C05494=1175.182,115.152,-52.912,-178.804,6.300,148.789
C05495=1175.178,115.401,-52.932,-178.801,6.302,148.788
C05496=1175.172,115.650,-52.951,-178.799,6.303,148.788
C05497=1175.168,115.900,-52.970,-178.796,6.304,148.787
C05498=1175.163,116.148,-52.989,-178.794,6.306,148.787
C05499=1175.158,116.398,-53.009,-178.790,6.307,148.786
C05500=1175.154,116.646,-53.028,-178.788,6.308,148.786
C05501=1175.149,116.897,-53.047,-178.786,6.310,148.785
C05502=1175.143,117.146,-53.066,-178.782,6.311,148.785
C05503=1175.139,117.395,-53.085,-178.780,6.312,148.784
C05504=1175.134,117.644,-53.105,-178.778,6.314,148.784
C05505=1175.129,117.893,-53.124,-178.775,6.316,148.784
C05506=1175.125,118.143,-53.143,-178.772,6.317,148.783
C05507=1175.120,118.391,-53.162,-178.770,6.318,148.783
C05508=1175.115,118.641,-53.182,-178.767,6.320,148.782
C05509=1175.110,118.890,-53.201,-178.764,6.322,148.782
C05510=1175.106,119.139,-53.220,-178.761,6.323,148.781
C05511=1175.101,119.389,-53.240,-178.759,6.324,148.781
C05512=1175.096,119.638,-53.259,-178.756,6.326,148.780
C05513=1175.091,119.887,-53.279,-178.753,6.327,148.780
C05514=1175.086,120.136,-53.298,-178.751,6.328,148.779
C05515=1175.082,120.385,-53.317,-178.748,6.330,148.779
C05516=1175.077,120.635,-53.337,-178.745,6.331,148.778
C05517=1175.071,120.884,-53.356,-178.743,6.333,148.778
C05518=1175.067,121.133,-53.376,-178.740,6.334,148.777
C05519=1175.062,121.382,-53.394,-178.737,6.335,148.777
C05520=1175.057,121.631,-53.414,-178.735,6.337,148.777
C05521=1175.053,121.880,-53.434,-178.732,6.339,148.776
C05522=1175.048,122.129,-53.454,-178.729,6.339,148.776
C05523=1175.043,122.379,-53.473,-178.727,6.341,148.775
C05524=1175.039,122.628,-53.492,-178.724,6.343,148.775
C05525=1175.033,122.877,-53.512,-178.721,6.345,148.774
C05526=1175.029,123.126,-53.531,-178.719,6.345,148.774
C05527=1175.024,123.376,-53.551,-178.716,6.347,148.773
C05528=1175.019,123.624,-53.571,-178.713,6.349,148.773
C05529=1175.014,123.874,-53.591,-178.711,6.350,148.773
C05530=1175.009,124.123,-53.610,-178.708,6.352,148.772
C05531=1175.004,124.372,-53.630,-178.705,6.353,148.772
C05532=1175.000,124.621,-53.649,-178.703,6.354,148.771
C05533=1174.996,124.870,-53.669,-178.700,6.356,148.771
C05534=1174.990,125.119,-53.688,-178.697,6.358,148.770
C05535=1174.986,125.369,-53.708,-178.694,6.358,148.770
C05536=1174.981,125.618,-53.728,-178.692,6.360,148.769
C05537=1174.976,125.867,-53.748,-178.689,6.362,148.769
C05538=1174.971,126.116,-53.767,-178.686,6.364,148.769
C05539=1174.966,126.366,-53.787,-178.684,6.365,148.768
C05540=1174.962,126.615,-53.807,-178.681,6.366,148.768
C05541=1174.957,126.864,-53.827,-178.678,6.368,148.767
C05542=1174.952,127.113,-53.846,-178.676,6.369,148.767
C05543=1174.947,127.363,-53.866,-178.673,6.371,148.766
C05544=1174.943,127.612,-53.886,-178.670,6.372,148.766
C05545=1174.937,127.861,-53.906,-178.668,6.374,148.765
C05546=1174.933,128.110,-53.926,-178.665,6.375,148.765
C05547=1174.928,128.359,-53.946,-178.662,6.377,148.765
C05548=1174.923,128.609,-53.965,-178.660,6.379,148.764
C05549=1174.918,128.857,-53.985,-178.657,6.379,148.763
C05550=1174.914,129.106,-54.005,-178.654,6.381,148.763
C05551=1174.909,129.356,-54.025,-178.652,6.383,148.763
C05552=1174.904,129.605,-54.045,-178.649,6.385,148.762
C05553=1174.900,129.855,-54.065,-178.646,6.386,148.762
C05554=1174.895,130.103,-54.085,-178.644,6.387,148.761
C05555=1174.890,130.352,-54.104,-178.641,6.389,148.761
C05556=1174.885,130.601,-54.125,-178.638,6.390,148.760
C05557=1174.881,130.851,-54.144,-178.635,6.392,148.760
C05558=1174.876,131.099,-54.164,-178.633,6.394,148.760
C05559=1174.871,131.349,-54.184,-178.631,6.395,148.759
C05560=1174.866,131.598,-54.204,-178.627,6.396,148.759
C05561=1174.861,131.848,-54.225,-178.625,6.398,148.758
C05562=1174.856,132.116,-54.247,-178.622,6.400,148.758
C05563=1174.851,132.385,-54.268,-178.619,6.401,148.757
C05564=1174.846,132.653,-54.289,-178.616,6.403,148.757
C05565=1174.841,132.921,-54.311,-178.613,6.404,148.757
C05566=1174.836,133.171,-54.331,-178.611,6.406,148.756
C05567=1174.831,133.420,-54.352,-178.608,6.408,148.756
C05568=1174.826,133.669,-54.371,-178.605,6.409,148.755
C05569=1174.821,133.918,-54.391,-178.603,6.410,148.755
C05570=1174.817,134.167,-54.412,-178.600,6.412,148.754
C05571=1174.812,134.416,-54.431,-178.597,6.414,148.754
C05572=1174.807,134.666,-54.452,-178.595,6.415,148.754
C05573=1174.803,134.915,-54.473,-178.591,6.417,148.753
C05574=1174.798,135.164,-54.492,-178.589,6.419,148.753
C05575=1174.794,135.413,-54.513,-178.586,6.420,148.752
C05576=1174.788,135.661,-54.533,-178.584,6.421,148.752
C05577=1174.783,135.911,-54.553,-178.581,6.423,148.751
C05578=1174.779,136.160,-54.573,-178.579,6.425,148.751
C05579=1174.774,136.409,-54.594,-178.575,6.426,148.750
C05580=1174.769,136.659,-54.613,-178.573,6.428,148.750
C05581=1174.764,136.908,-54.634,-178.570,6.430,148.750
C05582=1174.760,137.157,-54.655,-178.568,6.431,148.749
C05583=1174.755,137.406,-54.675,-178.565,6.432,148.749
C05584=1174.751,137.655,-54.695,-178.562,6.434,148.748
C05585=1174.745,137.905,-54.716,-178.560,6.436,148.748
C05586=1174.741,138.154,-54.736,-178.557,6.437,148.747
C05587=1174.737,138.403,-54.756,-178.554,6.439,148.747
C05588=1174.731,138.652,-54.777,-178.551,6.441,148.747
C05589=1174.726,138.901,-54.797,-178.549,6.442,148.746
C05590=1174.722,139.150,-54.817,-178.546,6.443,148.746
C05591=1174.716,139.399,-54.838,-178.544,6.445,148.745
C05592=1174.712,139.648,-54.858,-178.541,6.447,148.745
C05593=1174.708,139.897,-54.879,-178.538,6.448,148.744
C05594=1174.702,140.146,-54.900,-178.535,6.450,148.744
C05595=1174.698,140.395,-54.920,-178.532,6.452,148.744
C05596=1174.693,140.645,-54.940,-178.530,6.453,148.743
C05597=1174.688,140.894,-54.961,-178.528,6.454,148.743
C05598=1174.684,141.143,-54.981,-178.525,6.456,148.743
C05599=1174.679,141.392,-55.002,-178.522,6.458,148.742
C05600=1174.674,141.641,-55.023,-178.519,6.460,148.742
C05601=1174.670,141.890,-55.043,-178.517,6.461,148.741
C05602=1174.664,142.139,-55.064,-178.514,6.463,148.741
C05603=1174.660,142.388,-55.084,-178.511,6.465,148.740
C05604=1174.655,142.637,-55.105,-178.508,6.466,148.740
C05605=1174.650,142.886,-55.126,-178.505,6.468,148.740
C05606=1174.646,143.135,-55.146,-178.503,6.469,148.739
C05607=1174.641,143.385,-55.167,-178.501,6.471,148.739
C05608=1174.636,143.634,-55.187,-178.498,6.472,148.738
C05609=1174.631,143.883,-55.208,-178.495,6.474,148.738
C05610=1174.627,144.132,-55.229,-178.493,6.476,148.738
C05611=1174.622,144.382,-55.250,-178.489,6.477,148.737
C05612=1174.618,144.631,-55.270,-178.487,6.479,148.737
C05613=1174.612,144.880,-55.291,-178.484,6.481,148.736
C05614=1174.608,145.128,-55.312,-178.481,6.483,148.736
C05615=1174.603,145.378,-55.333,-178.479,6.484,148.736
C05616=1174.599,145.626,-55.354,-178.477,6.485,148.735
C05617=1174.594,145.876,-55.375,-178.474,6.487,148.735
C05618=1174.589,146.125,-55.395,-178.471,6.489,148.734
C05619=1174.584,146.374,-55.416,-178.468,6.491,148.734
C05620=1174.579,146.623,-55.436,-178.466,6.492,148.734
C05621=1174.574,146.872,-55.457,-178.463,6.494,148.733
C05622=1174.571,147.121,-55.479,-178.460,6.495,148.733
C05623=1174.566,147.370,-55.500,-178.457,6.497,148.732
C05624=1174.561,147.619,-55.520,-178.454,6.499,148.732
C05625=1174.556,147.869,-55.541,-178.452,6.501,148.731
C05626=1174.551,148.118,-55.562,-178.449,6.502,148.731
C05627=1174.547,148.366,-55.583,-178.446,6.504,148.731
C05628=1174.542,148.615,-55.604,-178.444,6.506,148.730
C05629=1174.537,148.864,-55.624,-178.442,6.507,148.730
C05630=1174.532,149.114,-55.645,-178.439,6.509,148.730
C05631=1174.528,149.363,-55.668,-178.436,6.510,148.729
C05632=1174.523,149.612,-55.688,-178.433,6.512,148.729
C05633=1174.518,149.861,-55.709,-178.431,6.514,148.728
C05634=1174.514,150.110,-55.730,-178.428,6.516,148.728
C05635=1174.509,150.359,-55.751,-178.425,6.517,148.727
C05636=1174.504,150.608,-55.772,-178.422,6.519,148.727
C05637=1174.500,150.857,-55.793,-178.420,6.521,148.727
C05638=1174.495,151.106,-55.814,-178.417,6.522,148.726
C05639=1174.490,151.356,-55.835,-178.414,6.524,148.726
C05640=1174.485,151.604,-55.857,-178.411,6.526,148.726
C05641=1174.480,151.853,-55.877,-178.409,6.528,148.725
C05642=1174.476,152.103,-55.899,-178.406,6.529,148.725
C05643=1174.471,152.352,-55.920,-178.403,6.531,148.724
C05644=1174.466,152.601,-55.941,-178.401,6.533,148.724
C05645=1174.462,152.849,-55.962,-178.398,6.535,148.724
C05646=1174.456,153.099,-55.983,-178.395,6.536,148.723
C05647=1174.452,153.348,-56.005,-178.393,6.538,148.723
C05648=1174.448,153.597,-56.026,-178.390,6.540,148.722
C05649=1174.443,153.846,-56.047,-178.387,6.542,148.722
C05650=1174.438,154.095,-56.068,-178.385,6.543,148.722
C05651=1174.433,154.343,-56.090,-178.382,6.544,148.721
C05652=1174.429,154.593,-56.111,-178.380,6.546,148.721
C05653=1174.424,154.842,-56.133,-178.377,6.548,148.721
C05654=1174.419,155.091,-56.153,-178.374,6.550,148.720
C05655=1174.414,155.340,-56.175,-178.372,6.551,148.720
C05656=1174.409,155.590,-56.197,-178.369,6.553,148.719
C05657=1174.405,155.838,-56.218,-178.366,6.555,148.719
C05658=1174.400,156.087,-56.239,-178.363,6.556,148.718
C05659=1174.396,156.337,-56.261,-178.360,6.558,148.718
C05660=1174.391,156.586,-56.282,-178.358,6.560,148.718
C05661=1174.386,156.834,-56.303,-178.355,6.562,148.717
C05662=1174.381,157.083,-56.325,-178.352,6.563,148.717
C05663=1174.377,157.333,-56.346,-178.350,6.565,148.717
C05664=1174.372,157.581,-56.367,-178.347,6.567,148.716
C05665=1174.367,157.830,-56.389,-178.344,6.569,148.716
C05666=1174.362,158.099,-56.412,-178.341,6.571,148.716
C05667=1174.357,158.368,-56.435,-178.338,6.573,148.715
C05668=1174.352,158.638,-56.459,-178.336,6.575,148.715
C05669=1174.347,158.906,-56.482,-178.333,6.576,148.714
C05670=1174.342,159.156,-56.503,-178.330,6.578,148.714
C05671=1174.338,159.405,-56.525,-178.328,6.580,148.714
C05672=1174.333,159.653,-56.547,-178.325,6.582,148.713
C05673=1174.328,159.902,-56.568,-178.322,6.583,148.713
C05674=1174.324,160.152,-56.590,-178.320,6.585,148.713
C05675=1174.319,160.401,-56.611,-178.317,6.587,148.712
C05676=1174.314,160.649,-56.633,-178.314,6.589,148.712
C05677=1174.310,160.899,-56.655,-178.311,6.590,148.711
C05678=1174.305,161.147,-56.677,-178.309,6.592,148.711
C05679=1174.300,161.397,-56.698,-178.306,6.594,148.711
C05680=1174.295,161.646,-56.720,-178.303,6.596,148.710
C05681=1174.290,161.895,-56.742,-178.301,6.598,148.710
C05682=1174.286,162.144,-56.764,-178.298,6.599,148.710
C05683=1174.281,162.393,-56.785,-178.295,6.602,148.709
C05684=1174.277,162.642,-56.807,-178.292,6.604,148.709
C05685=1174.272,162.891,-56.828,-178.289,6.605,148.708
C05686=1174.267,163.140,-56.850,-178.287,6.607,148.708
C05687=1174.263,163.389,-56.872,-178.284,6.609,148.708
C05688=1174.258,163.638,-56.894,-178.281,6.611,148.707
C05689=1174.253,163.887,-56.916,-178.279,6.612,148.707
C05690=1174.249,164.136,-56.937,-178.276,6.614,148.707
C05691=1174.244,164.384,-56.959,-178.273,6.616,148.706
C05692=1174.239,164.634,-56.981,-178.271,6.618,148.706
C05693=1174.235,164.882,-57.003,-178.268,6.619,148.705
C05694=1174.230,165.132,-57.025,-178.265,6.621,148.705
C05695=1174.225,165.380,-57.047,-178.263,6.623,148.705
C05696=1174.221,165.630,-57.069,-178.260,6.625,148.704
C05697=1174.216,165.878,-57.090,-178.257,6.627,148.704
C05698=1174.211,166.128,-57.113,-178.254,6.628,148.704
C05699=1174.206,166.377,-57.135,-178.252,6.630,148.703
C05700=1174.202,166.626,-57.157,-178.249,6.632,148.703
C05701=1174.197,166.875,-57.178,-178.247,6.634,148.703
C05702=1174.193,167.124,-57.200,-178.244,6.636,148.702
C05703=1174.188,167.373,-57.222,-178.242,6.637,148.702
C05704=1174.184,167.622,-57.244,-178.238,6.640,148.702
C05705=1174.178,167.871,-57.266,-178.236,6.642,148.701
C05706=1174.174,168.120,-57.288,-178.233,6.644,148.701
C05707=1174.169,168.369,-57.310,-178.230,6.645,148.701
C05708=1174.165,168.618,-57.333,-178.228,6.647,148.700
C05709=1174.160,168.866,-57.355,-178.225,6.649,148.700
C05710=1174.155,169.116,-57.377,-178.222,6.651,148.699
C05711=1174.150,169.365,-57.399,-178.219,6.652,148.699
C05712=1174.146,169.614,-57.421,-178.217,6.654,148.699
C05713=1174.141,169.863,-57.443,-178.214,6.656,148.698
C05714=1174.137,170.112,-57.466,-178.211,6.658,148.698
C05715=1174.132,170.360,-57.488,-178.209,6.659,148.698
C05716=1174.127,170.610,-57.510,-178.207,6.662,148.697
C05717=1174.123,170.858,-57.531,-178.203,6.664,148.697
C05718=1174.118,171.107,-57.555,-178.201,6.666,148.697
C05719=1174.113,171.356,-57.576,-178.198,6.668,148.696
C05720=1174.109,171.605,-57.598,-178.195,6.669,148.696
C05721=1174.104,171.855,-57.621,-178.193,6.671,148.696
C05722=1174.099,172.103,-57.644,-178.190,6.673,148.695
C05723=1174.095,172.352,-57.666,-178.187,6.675,148.695
C05724=1174.089,172.601,-57.688,-178.185,6.676,148.695
C05725=1174.085,172.850,-57.711,-178.182,6.678,148.694
C05726=1174.081,173.099,-57.733,-178.179,6.680,148.694
C05727=1174.075,173.348,-57.755,-178.176,6.683,148.694
C05728=1174.072,173.597,-57.778,-178.174,6.685,148.693
C05729=1174.067,173.846,-57.799,-178.171,6.686,148.693
C05730=1174.062,174.095,-57.822,-178.168,6.688,148.693
C05731=1174.058,174.344,-57.845,-178.166,6.690,148.692
C05732=1174.053,174.593,-57.866,-178.163,6.692,148.692
C05733=1174.048,174.842,-57.890,-178.160,6.694,148.692
C05734=1174.044,175.091,-57.912,-178.158,6.695,148.691
C05735=1174.038,175.340,-57.934,-178.155,6.697,148.691
C05736=1174.034,175.589,-57.957,-178.152,6.700,148.691
C05737=1174.029,175.837,-57.979,-178.149,6.702,148.690
C05738=1174.025,176.086,-58.002,-178.147,6.704,148.690
C05739=1174.020,176.336,-58.024,-178.144,6.705,148.690
C05740=1174.015,176.584,-58.047,-178.141,6.707,148.689
C05741=1174.011,176.833,-58.069,-178.139,6.709,148.689
C05742=1174.006,177.082,-58.092,-178.136,6.711,148.688
C05743=1174.002,177.332,-58.114,-178.133,6.713,148.688
C05744=1173.997,177.580,-58.137,-178.131,6.715,148.688
C05745=1173.992,177.829,-58.159,-178.128,6.717,148.688
C05746=1173.988,178.078,-58.182,-178.125,6.719,148.687
C05747=1173.983,178.326,-58.205,-178.123,6.721,148.687
C05748=1173.979,178.576,-58.227,-178.120,6.722,148.687
C05749=1173.974,178.825,-58.251,-178.117,6.724,148.686
C05750=1173.969,179.074,-58.273,-178.114,6.727,148.686
C05751=1173.965,179.322,-58.296,-178.111,6.729,148.685
C05752=1173.960,179.571,-58.319,-178.109,6.731,148.685
C05753=1173.956,179.821,-58.341,-178.106,6.732,148.685
C05754=1173.950,180.069,-58.364,-178.104,6.734,148.685
C05755=1173.946,180.318,-58.387,-178.101,6.736,148.684
C05756=1173.941,180.568,-58.410,-178.098,6.738,148.684
C05757=1173.937,180.816,-58.432,-178.095,6.740,148.684
C05758=1173.932,181.065,-58.455,-178.093,6.742,148.683
C05759=1173.928,181.314,-58.477,-178.090,6.744,148.683
C05760=1173.923,181.563,-58.501,-178.088,6.746,148.683
C05761=1173.918,181.812,-58.524,-178.085,6.748,148.682
C05762=1173.914,182.060,-58.546,-178.082,6.750,148.682
C05763=1173.909,182.310,-58.569,-178.079,6.752,148.682
C05764=1173.905,182.558,-58.592,-178.077,6.754,148.682
C05765=1173.900,182.807,-58.615,-178.074,6.756,148.681
C05766=1173.895,183.056,-58.639,-178.071,6.758,148.681
C05767=1173.891,183.304,-58.661,-178.069,6.760,148.680
C05768=1173.886,183.554,-58.684,-178.066,6.761,148.680
C05769=1173.881,183.803,-58.707,-178.063,6.764,148.680
C05770=1173.877,184.073,-58.731,-178.060,6.766,148.679
C05771=1173.871,184.342,-58.756,-178.057,6.768,148.679
C05772=1173.866,184.612,-58.781,-178.054,6.770,148.679
C05773=1173.862,184.881,-58.807,-178.052,6.772,148.679
C05774=1173.857,185.130,-58.830,-178.049,6.775,148.678
C05775=1173.852,185.380,-58.853,-178.046,6.777,148.678
C05776=1173.848,185.628,-58.875,-178.043,6.778,148.678
C05777=1173.843,185.877,-58.898,-178.041,6.780,148.677
C05778=1173.838,186.126,-58.922,-178.038,6.782,148.677
C05779=1173.833,186.375,-58.945,-178.035,6.785,148.677
C05780=1173.829,186.623,-58.968,-178.033,6.787,148.676
C05781=1173.825,186.872,-58.991,-178.030,6.788,148.676
C05782=1173.820,187.122,-59.015,-178.027,6.790,148.676
C05783=1173.815,187.371,-59.038,-178.025,6.792,148.676
C05784=1173.811,187.619,-59.061,-178.022,6.795,148.675
C05785=1173.806,187.868,-59.084,-178.019,6.797,148.675
C05786=1173.801,188.117,-59.107,-178.016,6.798,148.674
C05787=1173.797,188.366,-59.130,-178.014,6.800,148.674
C05788=1173.792,188.615,-59.154,-178.011,6.803,148.674
C05789=1173.787,188.864,-59.177,-178.008,6.805,148.674
C05790=1173.783,189.112,-59.200,-178.006,6.807,148.673
C05791=1173.779,189.361,-59.223,-178.003,6.808,148.673
C05792=1173.774,189.611,-59.247,-178.000,6.810,148.673
C05793=1173.769,189.859,-59.271,-177.997,6.813,148.672
C05794=1173.765,190.108,-59.294,-177.995,6.815,148.672
C05795=1173.760,190.357,-59.317,-177.992,6.817,148.672
C05796=1173.755,190.605,-59.340,-177.989,6.819,148.671
C05797=1173.751,190.854,-59.363,-177.987,6.821,148.671
C05798=1173.746,191.103,-59.387,-177.984,6.823,148.671
C05799=1173.741,191.352,-59.410,-177.981,6.825,148.671
C05800=1173.737,191.601,-59.434,-177.979,6.827,148.670
C05801=1173.732,191.850,-59.457,-177.976,6.829,148.670
C05802=1173.728,192.099,-59.481,-177.973,6.832,148.670
C05803=1173.723,192.348,-59.504,-177.971,6.833,148.669
C05804=1173.718,192.596,-59.528,-177.968,6.835,148.669
C05805=1173.714,192.845,-59.551,-177.966,6.837,148.669
C05806=1173.709,193.094,-59.575,-177.962,6.840,148.669
C05807=1173.704,193.343,-59.598,-177.960,6.842,148.668
C05808=1173.700,193.592,-59.622,-177.957,6.843,148.668
C05809=1173.695,193.841,-59.646,-177.955,6.845,148.668
C05810=1173.691,194.090,-59.669,-177.952,6.848,148.667
C05811=1173.686,194.339,-59.692,-177.949,6.850,148.667
C05812=1173.682,194.587,-59.716,-177.946,6.852,148.667
C05813=1173.677,194.836,-59.740,-177.944,6.854,148.667
C05814=1173.672,195.084,-59.764,-177.941,6.856,148.666
C05815=1173.668,195.334,-59.787,-177.938,6.858,148.666
C05816=1173.663,195.583,-59.811,-177.936,6.860,148.666
C05817=1173.659,195.831,-59.835,-177.933,6.863,148.665
C05818=1173.654,196.080,-59.858,-177.930,6.865,148.665
C05819=1173.649,196.329,-59.881,-177.927,6.866,148.665
C05820=1173.645,196.577,-59.905,-177.925,6.868,148.664
C05821=1173.641,196.827,-59.929,-177.922,6.871,148.664
C05822=1173.636,197.076,-59.953,-177.919,6.873,148.664
C05823=1173.632,197.325,-59.977,-177.917,6.875,148.664
C05824=1173.627,197.573,-60.001,-177.914,6.877,148.664
C05825=1173.623,197.822,-60.024,-177.911,6.879,148.663
C05826=1173.617,198.071,-60.049,-177.909,6.881,148.663
C05827=1173.613,198.320,-60.072,-177.906,6.883,148.662
C05828=1173.608,198.568,-60.096,-177.903,6.886,148.662
C05829=1173.604,198.817,-60.119,-177.900,6.888,148.662
C05830=1173.599,199.066,-60.144,-177.898,6.889,148.662
C05831=1173.595,199.315,-60.167,-177.896,6.892,148.662
C05832=1173.591,199.564,-60.191,-177.892,6.894,148.661
C05833=1173.585,199.813,-60.215,-177.890,6.896,148.661
C05834=1173.581,200.062,-60.239,-177.887,6.898,148.661
C05835=1173.576,200.310,-60.263,-177.884,6.901,148.660
C05836=1173.572,200.559,-60.287,-177.882,6.903,148.660
C05837=1173.567,200.807,-60.311,-177.879,6.904,148.660
C05838=1173.563,201.056,-60.335,-177.876,6.907,148.660
C05839=1173.558,201.306,-60.359,-177.873,6.909,148.659
C05840=1173.554,201.554,-60.383,-177.871,6.911,148.659
C05841=1173.549,201.803,-60.407,-177.869,6.913,148.659
C05842=1173.545,202.052,-60.431,-177.865,6.916,148.659
C05843=1173.540,202.300,-60.455,-177.863,6.917,148.658
C05844=1173.535,202.549,-60.480,-177.860,6.919,148.658
C05845=1173.531,202.799,-60.503,-177.857,6.922,148.658
C05846=1173.527,203.047,-60.527,-177.855,6.924,148.657
C05847=1173.522,203.296,-60.552,-177.852,6.926,148.657
C05848=1173.517,203.544,-60.576,-177.849,6.929,148.657
C05849=1173.512,203.793,-60.599,-177.846,6.930,148.657
C05850=1173.509,204.042,-60.624,-177.844,6.932,148.656
C05851=1173.504,204.291,-60.649,-177.841,6.935,148.656
C05852=1173.499,204.539,-60.673,-177.838,6.937,148.656
C05853=1173.495,204.788,-60.697,-177.836,6.939,148.656
C05854=1173.489,205.037,-60.721,-177.833,6.942,148.655
C05855=1173.485,205.286,-60.745,-177.830,6.943,148.655
C05856=1173.481,205.535,-60.769,-177.828,6.946,148.655
C05857=1173.476,205.783,-60.794,-177.825,6.948,148.655
C05858=1173.472,206.032,-60.818,-177.822,6.950,148.654
C05859=1173.467,206.281,-60.843,-177.820,6.952,148.654
C05860=1173.463,206.530,-60.867,-177.817,6.955,148.654
C05861=1173.458,206.779,-60.890,-177.814,6.957,148.654
C05862=1173.453,207.027,-60.915,-177.812,6.959,148.653
C05863=1173.449,207.277,-60.939,-177.809,6.961,148.653
C05864=1173.444,207.525,-60.964,-177.806,6.963,148.653
C05865=1173.439,207.774,-60.988,-177.804,6.965,148.653
C05866=1173.436,208.023,-61.013,-177.800,6.968,148.652
C05867=1173.431,208.272,-61.037,-177.798,6.970,148.652
C05868=1173.426,208.520,-61.061,-177.796,6.972,148.652
C05869=1173.421,208.769,-61.086,-177.792,6.974,148.651
C05870=1173.417,209.018,-61.111,-177.790,6.976,148.651
C05871=1173.412,209.267,-61.135,-177.787,6.979,148.651
C05872=1173.408,209.515,-61.159,-177.785,6.981,148.651
C05873=1173.403,209.764,-61.184,-177.782,6.983,148.651
C05874=1173.398,210.035,-61.211,-177.779,6.985,148.650
C05875=1173.393,210.305,-61.238,-177.776,6.988,148.650
C05876=1173.389,210.575,-61.264,-177.773,6.990,148.650
C05877=1173.384,210.845,-61.291,-177.770,6.993,148.649
C05878=1173.379,211.094,-61.316,-177.768,6.995,148.649
C05879=1173.375,211.343,-61.340,-177.765,6.998,148.649
C05880=1173.370,211.592,-61.365,-177.762,6.999,148.649
C05881=1173.365,211.841,-61.389,-177.760,7.001,148.649
C05882=1173.361,212.090,-61.414,-177.757,7.004,148.648
C05883=1173.356,212.338,-61.439,-177.754,7.006,148.648
C05884=1173.352,212.587,-61.464,-177.751,7.009,148.648
C05885=1173.347,212.836,-61.488,-177.749,7.011,148.648
C05886=1173.343,213.084,-61.512,-177.746,7.013,148.647
C05887=1173.338,213.334,-61.537,-177.743,7.015,148.647
C05888=1173.333,213.582,-61.563,-177.741,7.017,148.647
C05889=1173.329,213.830,-61.587,-177.738,7.020,148.647
C05890=1173.325,214.080,-61.612,-177.735,7.022,148.646
C05891=1173.319,214.328,-61.637,-177.733,7.024,148.646
C05892=1173.316,214.577,-61.662,-177.730,7.027,148.646
C05893=1173.311,214.826,-61.686,-177.727,7.029,148.646
C05894=1173.307,215.075,-61.711,-177.724,7.031,148.645
C05895=1173.302,215.323,-61.736,-177.722,7.033,148.645
C05896=1173.297,215.571,-61.761,-177.719,7.035,148.645
C05897=1173.293,215.821,-61.785,-177.716,7.038,148.645
C05898=1173.288,216.069,-61.811,-177.714,7.040,148.645
C05899=1173.284,216.318,-61.836,-177.711,7.043,148.644
C05900=1173.279,216.567,-61.860,-177.709,7.045,148.644
C05901=1173.275,216.815,-61.886,-177.706,7.047,148.644
C05902=1173.270,217.064,-61.910,-177.703,7.049,148.644
C05903=1173.266,217.313,-61.936,-177.700,7.051,148.643
C05904=1173.262,217.561,-61.960,-177.697,7.054,148.643
C05905=1173.257,217.810,-61.986,-177.695,7.056,148.643
C05906=1173.252,218.059,-62.010,-177.692,7.059,148.643
C05907=1173.248,218.308,-62.036,-177.690,7.061,148.643
C05908=1173.244,218.556,-62.060,-177.687,7.063,148.642
C05909=1173.239,218.805,-62.085,-177.684,7.066,148.642
C05910=1173.234,219.054,-62.111,-177.682,7.067,148.642
C05911=1173.230,219.303,-62.136,-177.678,7.070,148.641
C05912=1173.226,219.551,-62.161,-177.676,7.072,148.641
C05913=1173.221,219.800,-62.186,-177.673,7.075,148.641
C05914=1173.216,220.048,-62.211,-177.671,7.077,148.641
C05915=1173.212,220.297,-62.237,-177.668,7.079,148.641
C05916=1173.207,220.546,-62.261,-177.665,7.082,148.641
C05917=1173.203,220.795,-62.287,-177.663,7.083,148.640
C05918=1173.198,221.043,-62.311,-177.660,7.086,148.640
C05919=1173.194,221.292,-62.337,-177.657,7.088,148.640
C05920=1173.189,221.540,-62.362,-177.654,7.091,148.640
C05921=1173.185,221.789,-62.387,-177.652,7.093,148.639
C05922=1173.180,222.038,-62.413,-177.649,7.096,148.639
C05923=1173.176,222.286,-62.439,-177.646,7.098,148.639
C05924=1173.171,222.536,-62.464,-177.644,7.101,148.639
C05925=1173.166,222.784,-62.489,-177.641,7.102,148.639
C05926=1173.163,223.032,-62.514,-177.639,7.104,148.638
C05927=1173.158,223.281,-62.539,-177.635,7.107,148.638
C05928=1173.153,223.530,-62.565,-177.633,7.109,148.638
C05929=1173.149,223.779,-62.590,-177.630,7.112,148.638
C05930=1173.144,224.027,-62.616,-177.628,7.114,148.638
C05931=1173.140,224.276,-62.641,-177.625,7.117,148.637
C05932=1173.136,224.525,-62.666,-177.622,7.119,148.637
C05933=1173.131,224.773,-62.692,-177.619,7.121,148.637
C05934=1173.127,225.022,-62.718,-177.617,7.123,148.637
C05935=1173.122,225.270,-62.743,-177.614,7.126,148.636
C05936=1173.117,225.519,-62.768,-177.612,7.128,148.636
C05937=1173.113,225.768,-62.794,-177.608,7.131,148.636
C05938=1173.108,226.016,-62.819,-177.606,7.133,148.636
C05939=1173.104,226.265,-62.845,-177.603,7.136,148.636
C05940=1173.100,226.514,-62.871,-177.601,7.138,148.636
C05941=1173.095,226.762,-62.896,-177.598,7.140,148.635
C05942=1173.091,227.011,-62.922,-177.595,7.142,148.635
C05943=1173.086,227.260,-62.947,-177.592,7.145,148.635
C05944=1173.081,227.508,-62.972,-177.590,7.147,148.635
C05945=1173.077,227.757,-62.998,-177.587,7.150,148.635
C05946=1173.073,228.006,-63.024,-177.585,7.152,148.634
C05947=1173.068,228.254,-63.049,-177.582,7.155,148.634
C05948=1173.063,228.503,-63.075,-177.579,7.157,148.634
C05949=1173.059,228.752,-63.101,-177.576,7.160,148.634
C05950=1173.054,229.000,-63.127,-177.574,7.162,148.633
C05951=1173.050,229.249,-63.152,-177.571,7.164,148.633
C05952=1173.046,229.498,-63.178,-177.568,7.166,148.633
C05953=1173.041,229.746,-63.204,-177.566,7.169,148.633
C05954=1173.036,229.995,-63.229,-177.563,7.171,148.633
C05955=1173.032,230.243,-63.255,-177.560,7.174,148.633
C05956=1173.027,230.493,-63.281,-177.558,7.176,148.632
C05957=1173.023,230.741,-63.307,-177.555,7.179,148.632
C05958=1173.018,230.989,-63.332,-177.553,7.181,148.632
C05959=1173.014,231.238,-63.359,-177.549,7.183,148.632
C05960=1173.010,231.486,-63.385,-177.547,7.186,148.632
C05961=1173.006,231.735,-63.410,-177.544,7.189,148.632
C05962=1173.000,231.984,-63.436,-177.542,7.190,148.631
C05963=1172.996,232.232,-63.462,-177.539,7.193,148.631
C05964=1172.992,232.481,-63.488,-177.536,7.195,148.631
C05965=1172.988,232.730,-63.514,-177.534,7.198,148.631
C05966=1172.982,232.978,-63.540,-177.531,7.200,148.631
C05967=1172.978,233.227,-63.566,-177.528,7.203,148.630
C05968=1172.974,233.475,-63.592,-177.526,7.205,148.630
C05969=1172.970,233.724,-63.618,-177.523,7.208,148.630
C05970=1172.965,233.973,-63.645,-177.520,7.211,148.630
C05971=1172.960,234.221,-63.670,-177.518,7.213,148.630
C05972=1172.956,234.470,-63.696,-177.515,7.215,148.630
C05973=1172.952,234.718,-63.722,-177.512,7.217,148.629
C05974=1172.947,234.967,-63.749,-177.509,7.220,148.629
C05975=1172.943,235.216,-63.774,-177.507,7.222,148.629
C05976=1172.939,235.465,-63.800,-177.504,7.225,148.629
C05977=1172.933,235.712,-63.827,-177.502,7.227,148.629
C05978=1172.929,235.984,-63.855,-177.499,7.230,148.629
C05979=1172.924,236.256,-63.884,-177.496,7.233,148.628
C05980=1172.919,236.528,-63.912,-177.493,7.236,148.628
C05981=1172.915,236.799,-63.941,-177.490,7.238,148.628
C05982=1172.910,237.048,-63.967,-177.487,7.241,148.628
C05983=1172.905,237.297,-63.993,-177.485,7.243,148.628
C05984=1172.901,237.545,-64.020,-177.481,7.246,148.627
C05985=1172.896,237.794,-64.046,-177.479,7.248,148.627
C05986=1172.892,238.042,-64.072,-177.476,7.251,148.627
C05987=1172.888,238.291,-64.098,-177.474,7.253,148.627
C05988=1172.883,238.539,-64.125,-177.471,7.256,148.627
C05989=1172.879,238.788,-64.151,-177.468,7.258,148.627
C05990=1172.874,239.036,-64.178,-177.466,7.260,148.626
C05991=1172.870,239.285,-64.203,-177.463,7.263,148.626
C05992=1172.865,239.534,-64.230,-177.460,7.265,148.626
C05993=1172.861,239.782,-64.256,-177.458,7.268,148.626
C05994=1172.856,240.031,-64.283,-177.455,7.270,148.626
C05995=1172.852,240.280,-64.309,-177.452,7.273,148.626
C05996=1172.848,240.528,-64.336,-177.449,7.276,148.626
C05997=1172.843,240.777,-64.362,-177.447,7.278,148.625
C05998=1172.838,241.025,-64.389,-177.444,7.281,148.625
C05999=1172.834,241.273,-64.415,-177.442,7.283,148.625
C06000=1172.829,241.522,-64.441,-177.439,7.286,148.625
C06001=1172.825,241.770,-64.468,-177.436,7.289,148.625
C06002=1172.821,242.019,-64.495,-177.434,7.291,148.625
C06003=1172.816,242.268,-64.521,-177.431,7.294,148.625
C06004=1172.812,242.516,-64.548,-177.429,7.296,148.624
C06005=1172.808,242.764,-64.574,-177.425,7.298,148.624
C06006=1172.803,243.013,-64.600,-177.423,7.301,148.624
C06007=1172.799,243.262,-64.627,-177.421,7.303,148.624
C06008=1172.794,243.510,-64.654,-177.417,7.306,148.624
C06009=1172.789,243.759,-64.680,-177.415,7.308,148.624
C06010=1172.785,244.007,-64.707,-177.412,7.311,148.624
C06011=1172.781,244.256,-64.734,-177.410,7.314,148.623
C06012=1172.777,244.504,-64.760,-177.407,7.316,148.623
C06013=1172.772,244.753,-64.787,-177.404,7.319,148.623
C06014=1172.767,245.002,-64.814,-177.401,7.322,148.623
C06015=1172.763,245.250,-64.840,-177.399,7.324,148.623
C06016=1172.759,245.498,-64.867,-177.396,7.327,148.623
C06017=1172.754,245.747,-64.894,-177.394,7.329,148.622
C06018=1172.751,245.996,-64.921,-177.391,7.332,148.622
C06019=1172.746,246.245,-64.948,-177.388,7.334,148.622
C06020=1172.741,246.493,-64.975,-177.386,7.336,148.622
C06021=1172.737,246.742,-65.001,-177.383,7.339,148.622
C06022=1172.732,246.990,-65.028,-177.380,7.342,148.622
C06023=1172.728,247.239,-65.055,-177.378,7.344,148.622
C06024=1172.724,247.487,-65.082,-177.375,7.347,148.622
C06025=1172.719,247.735,-65.109,-177.372,7.350,148.621
C06026=1172.715,247.984,-65.136,-177.370,7.352,148.621
C06027=1172.710,248.232,-65.163,-177.367,7.355,148.621
C06028=1172.706,248.480,-65.189,-177.365,7.357,148.621
C06029=1172.701,248.729,-65.216,-177.362,7.360,148.621
C06030=1172.697,248.978,-65.244,-177.359,7.363,148.621
C06031=1172.693,249.227,-65.271,-177.357,7.365,148.621
C06032=1172.689,249.475,-65.297,-177.354,7.368,148.620
C06033=1172.684,249.723,-65.324,-177.351,7.371,148.620
C06034=1172.679,249.972,-65.351,-177.349,7.373,148.620
C06035=1172.675,250.220,-65.378,-177.346,7.376,148.620
C06036=1172.670,250.469,-65.406,-177.343,7.378,148.620
C06037=1172.665,250.717,-65.433,-177.341,7.381,148.620
C06038=1172.662,250.966,-65.459,-177.338,7.384,148.620
C06039=1172.657,251.215,-65.486,-177.335,7.387,148.620
C06040=1172.653,251.463,-65.514,-177.333,7.389,148.620
C06041=1172.648,251.712,-65.541,-177.330,7.391,148.619
C06042=1172.644,251.959,-65.568,-177.327,7.394,148.619
C06043=1172.639,252.208,-65.595,-177.325,7.396,148.619
C06044=1172.636,252.457,-65.622,-177.322,7.399,148.619
C06045=1172.631,252.705,-65.649,-177.319,7.402,148.619
C06046=1172.626,252.954,-65.676,-177.317,7.404,148.619
C06047=1172.622,253.202,-65.703,-177.314,7.407,148.619
C06048=1172.617,253.450,-65.731,-177.311,7.410,148.619
C06049=1172.613,253.699,-65.759,-177.309,7.412,148.619
C06050=1172.609,253.948,-65.786,-177.306,7.415,148.619
C06051=1172.604,254.196,-65.813,-177.303,7.418,148.618
C06052=1172.600,254.444,-65.841,-177.300,7.421,148.618
C06053=1172.596,254.694,-65.868,-177.298,7.423,148.618
C06054=1172.591,254.942,-65.895,-177.295,7.426,148.618
C06055=1172.587,255.190,-65.923,-177.293,7.429,148.618
C06056=1172.582,255.438,-65.950,-177.290,7.431,148.618
C06057=1172.578,255.688,-65.977,-177.288,7.434,148.618
C06058=1172.574,255.935,-66.005,-177.284,7.437,148.618
C06059=1172.569,256.184,-66.032,-177.282,7.439,148.617
C06060=1172.564,256.432,-66.059,-177.279,7.442,148.617
C06061=1172.561,256.681,-66.087,-177.277,7.445,148.617
C06062=1172.556,256.930,-66.114,-177.274,7.448,148.617
C06063=1172.552,257.177,-66.142,-177.272,7.450,148.617
C06064=1172.547,257.426,-66.169,-177.269,7.452,148.617
C06065=1172.543,257.675,-66.197,-177.266,7.455,148.617
C06066=1172.538,257.923,-66.224,-177.264,7.458,148.617
C06067=1172.534,258.171,-66.252,-177.261,7.460,148.617
C06068=1172.530,258.420,-66.280,-177.258,7.463,148.617
C06069=1172.525,258.669,-66.307,-177.256,7.466,148.617
C06070=1172.521,258.916,-66.335,-177.253,7.469,148.616
C06071=1172.517,259.166,-66.362,-177.250,7.472,148.616
C06072=1172.512,259.414,-66.390,-177.247,7.474,148.616
C06073=1172.507,259.662,-66.417,-177.245,7.476,148.616
C06074=1172.503,259.911,-66.446,-177.242,7.479,148.616
C06075=1172.499,260.159,-66.473,-177.240,7.482,148.616
C06076=1172.494,260.407,-66.500,-177.237,7.485,148.616
C06077=1172.491,260.656,-66.529,-177.235,7.487,148.616
C06078=1172.486,260.904,-66.556,-177.232,7.490,148.616
C06079=1172.481,261.152,-66.584,-177.229,7.493,148.616
C06080=1172.477,261.401,-66.612,-177.227,7.495,148.616
C06081=1172.473,261.650,-66.639,-177.224,7.498,148.616
C06082=1172.468,261.923,-66.670,-177.221,7.501,148.615
C06083=1172.463,262.195,-66.700,-177.218,7.504,148.615
C06084=1172.458,262.469,-66.731,-177.215,7.508,148.615
C06085=1172.453,262.742,-66.761,-177.212,7.511,148.615
C06086=1172.449,262.990,-66.789,-177.210,7.513,148.615
C06087=1172.445,263.239,-66.817,-177.207,7.516,148.615
C06088=1172.441,263.486,-66.845,-177.205,7.519,148.615
C06089=1172.435,263.735,-66.873,-177.201,7.521,148.615
C06090=1172.432,263.984,-66.901,-177.199,7.524,148.615
C06091=1172.427,264.232,-66.929,-177.196,7.527,148.615
C06092=1172.423,264.481,-66.958,-177.194,7.530,148.615
C06093=1172.419,264.729,-66.985,-177.191,7.533,148.614
C06094=1172.414,264.978,-67.013,-177.189,7.535,148.614
C06095=1172.410,265.226,-67.040,-177.186,7.538,148.614
C06096=1172.406,265.474,-67.069,-177.183,7.541,148.614
C06097=1172.401,265.722,-67.097,-177.181,7.544,148.614
C06098=1172.397,265.970,-67.125,-177.178,7.546,148.614
C06099=1172.392,266.219,-67.154,-177.176,7.549,148.614
C06100=1172.388,266.467,-67.181,-177.173,7.552,148.614
C06101=1172.383,266.716,-67.209,-177.170,7.555,148.614
C06102=1172.379,266.964,-67.237,-177.167,7.558,148.614
C06103=1172.375,267.213,-67.265,-177.165,7.560,148.614
C06104=1172.370,267.461,-67.294,-177.162,7.563,148.614
C06105=1172.366,267.710,-67.322,-177.160,7.566,148.614
C06106=1172.362,267.958,-67.350,-177.157,7.569,148.614
C06107=1172.358,268.206,-67.378,-177.155,7.571,148.614
C06108=1172.353,268.454,-67.406,-177.152,7.574,148.614
C06109=1172.349,268.703,-67.435,-177.149,7.577,148.613
C06110=1172.344,268.951,-67.463,-177.147,7.580,148.613
C06111=1172.340,269.200,-67.491,-177.144,7.583,148.613
C06112=1172.336,269.448,-67.519,-177.142,7.585,148.613
C06113=1172.331,269.697,-67.548,-177.139,7.588,148.613
C06114=1172.327,269.945,-67.576,-177.136,7.591,148.613
C06115=1172.322,270.194,-67.604,-177.133,7.594,148.613
C06116=1172.319,270.441,-67.633,-177.131,7.597,148.613
C06117=1172.314,270.689,-67.661,-177.128,7.599,148.613
C06118=1172.310,270.938,-67.690,-177.126,7.602,148.613
C06119=1172.305,271.186,-67.718,-177.123,7.605,148.613
C06120=1172.301,271.435,-67.746,-177.120,7.608,148.613
C06121=1172.296,271.683,-67.775,-177.118,7.610,148.613
C06122=1172.292,271.932,-67.803,-177.115,7.613,148.613
C06123=1172.288,272.180,-67.832,-177.113,7.616,148.613
C06124=1172.284,272.428,-67.860,-177.110,7.619,148.613
C06125=1172.279,272.677,-67.889,-177.107,7.622,148.613
C06126=1172.275,272.925,-67.916,-177.104,7.625,148.613
C06127=1172.271,273.173,-67.946,-177.102,7.627,148.612
C06128=1172.267,273.422,-67.974,-177.099,7.630,148.612
C06129=1172.262,273.670,-68.002,-177.097,7.633,148.612
C06130=1172.257,273.919,-68.031,-177.094,7.636,148.612
C06131=1172.253,274.166,-68.060,-177.091,7.639,148.612
C06132=1172.249,274.415,-68.088,-177.089,7.641,148.612
C06133=1172.244,274.664,-68.117,-177.086,7.644,148.612
C06134=1172.240,274.911,-68.146,-177.084,7.647,148.612
C06135=1172.236,275.160,-68.174,-177.081,7.650,148.612
C06136=1172.232,275.408,-68.203,-177.078,7.653,148.612
C06137=1172.227,275.656,-68.232,-177.075,7.656,148.612
C06138=1172.223,275.905,-68.260,-177.073,7.658,148.612
C06139=1172.219,276.153,-68.289,-177.070,7.661,148.612
C06140=1172.214,276.401,-68.318,-177.068,7.664,148.612
C06141=1172.210,276.650,-68.346,-177.065,7.667,148.612
C06142=1172.206,276.898,-68.376,-177.062,7.670,148.612
C06143=1172.201,277.146,-68.404,-177.060,7.672,148.612
C06144=1172.197,277.394,-68.433,-177.058,7.675,148.612
C06145=1172.193,277.643,-68.462,-177.055,7.678,148.612
C06146=1172.189,277.891,-68.491,-177.052,7.681,148.612
C06147=1172.184,278.139,-68.519,-177.049,7.684,148.612
C06148=1172.180,278.388,-68.548,-177.047,7.687,148.612
C06149=1172.175,278.636,-68.577,-177.044,7.690,148.612
C06150=1172.172,278.884,-68.606,-177.042,7.692,148.612
C06151=1172.167,279.133,-68.634,-177.039,7.695,148.612
C06152=1172.163,279.381,-68.664,-177.036,7.698,148.611
C06153=1172.158,279.629,-68.693,-177.034,7.701,148.611
C06154=1172.154,279.878,-68.722,-177.031,7.704,148.611
C06155=1172.150,280.125,-68.751,-177.029,7.707,148.612
C06156=1172.145,280.374,-68.779,-177.026,7.710,148.611
C06157=1172.141,280.622,-68.809,-177.024,7.713,148.611
C06158=1172.137,280.871,-68.838,-177.021,7.716,148.611
C06159=1172.132,281.119,-68.867,-177.018,7.719,148.611
C06160=1172.128,281.367,-68.896,-177.015,7.722,148.611
C06161=1172.124,281.615,-68.925,-177.013,7.724,148.611
C06162=1172.120,281.864,-68.954,-177.010,7.727,148.611
C06163=1172.115,282.112,-68.983,-177.008,7.730,148.611
C06164=1172.111,282.360,-69.012,-177.005,7.733,148.611
C06165=1172.107,282.608,-69.042,-177.003,7.736,148.611
C06166=1172.102,282.857,-69.070,-177.000,7.739,148.611
C06167=1172.098,283.105,-69.100,-176.997,7.742,148.611
C06168=1172.094,283.353,-69.129,-176.995,7.745,148.611
C06169=1172.089,283.601,-69.158,-176.992,7.748,148.611
C06170=1172.085,283.850,-69.187,-176.989,7.751,148.611
C06171=1172.080,284.098,-69.217,-176.987,7.753,148.611
C06172=1172.076,284.346,-69.246,-176.985,7.756,148.611
C06173=1172.072,284.595,-69.275,-176.982,7.759,148.611
C06174=1172.068,284.843,-69.305,-176.979,7.762,148.611
C06175=1172.063,285.091,-69.334,-176.976,7.765,148.611
C06176=1172.059,285.339,-69.363,-176.974,7.768,148.611
C06177=1172.054,285.588,-69.392,-176.971,7.771,148.611
C06178=1172.050,285.836,-69.422,-176.969,7.774,148.611
C06179=1172.046,286.084,-69.451,-176.966,7.777,148.611
C06180=1172.042,286.333,-69.481,-176.964,7.779,148.611
C06181=1172.038,286.581,-69.510,-176.961,7.782,148.611
C06182=1172.034,286.829,-69.539,-176.958,7.785,148.611
C06183=1172.029,287.077,-69.568,-176.955,7.788,148.611
C06184=1172.025,287.325,-69.598,-176.953,7.792,148.611
C06185=1172.020,287.573,-69.627,-176.950,7.795,148.611
C06186=1172.016,287.848,-69.661,-176.948,7.798,148.611
C06187=1172.012,288.123,-69.693,-176.945,7.801,148.611
C06188=1172.006,288.398,-69.725,-176.942,7.804,148.611
C06189=1172.001,288.672,-69.758,-176.939,7.807,148.611
C06190=1171.997,288.921,-69.788,-176.936,7.810,148.611
C06191=1171.993,289.169,-69.817,-176.934,7.814,148.611
C06192=1171.989,289.417,-69.847,-176.931,7.817,148.611
C06193=1171.985,289.666,-69.876,-176.928,7.820,148.611
C06194=1171.980,289.914,-69.906,-176.926,7.823,148.611
C06195=1171.977,290.161,-69.936,-176.924,7.825,148.611
C06196=1171.972,290.410,-69.966,-176.921,7.828,148.611
C06197=1171.967,290.658,-69.995,-176.919,7.831,148.611
C06198=1171.963,290.907,-70.025,-176.916,7.834,148.611
C06199=1171.959,291.155,-70.054,-176.913,7.837,148.611
C06200=1171.955,291.402,-70.084,-176.910,7.840,148.611
C06201=1171.950,291.651,-70.114,-176.908,7.843,148.611
C06202=1171.946,291.899,-70.144,-176.905,7.846,148.611
C06203=1171.942,292.148,-70.173,-176.903,7.849,148.611
C06204=1171.938,292.396,-70.203,-176.900,7.852,148.611
C06205=1171.934,292.643,-70.233,-176.898,7.855,148.611
C06206=1171.929,292.892,-70.263,-176.895,7.858,148.611
C06207=1171.925,293.140,-70.292,-176.893,7.861,148.611
C06208=1171.921,293.388,-70.323,-176.890,7.864,148.611
C06209=1171.916,293.637,-70.353,-176.887,7.867,148.611
C06210=1171.912,293.885,-70.382,-176.885,7.870,148.611
C06211=1171.908,294.132,-70.412,-176.882,7.873,148.611
C06212=1171.904,294.381,-70.442,-176.879,7.876,148.611
C06213=1171.899,294.629,-70.472,-176.877,7.879,148.611
C06214=1171.895,294.877,-70.502,-176.874,7.882,148.611
C06215=1171.891,295.125,-70.531,-176.872,7.885,148.611
C06216=1171.886,295.373,-70.562,-176.869,7.888,148.611
C06217=1171.883,295.622,-70.592,-176.866,7.891,148.611
C06218=1171.879,295.870,-70.622,-176.864,7.894,148.612
C06219=1171.874,296.118,-70.652,-176.861,7.897,148.611
C06220=1171.870,296.367,-70.682,-176.859,7.899,148.611
C06221=1171.866,296.614,-70.712,-176.857,7.903,148.612
C06222=1171.861,296.863,-70.742,-176.854,7.906,148.612
C06223=1171.857,297.111,-70.772,-176.851,7.909,148.612
C06224=1171.852,297.358,-70.803,-176.848,7.912,148.611
C06225=1171.848,297.607,-70.832,-176.846,7.915,148.612
C06226=1171.844,297.854,-70.862,-176.843,7.918,148.612
C06227=1171.840,298.104,-70.893,-176.841,7.921,148.612
C06228=1171.836,298.351,-70.923,-176.838,7.924,148.612
C06229=1171.831,298.600,-70.953,-176.836,7.927,148.612
C06230=1171.827,298.848,-70.983,-176.833,7.930,148.612
C06231=1171.823,299.095,-71.014,-176.830,7.933,148.612
C06232=1171.818,299.344,-71.043,-176.828,7.936,148.612
C06233=1171.814,299.592,-71.074,-176.825,7.939,148.612
C06234=1171.810,299.841,-71.104,-176.822,7.942,148.612
C06235=1171.806,300.089,-71.135,-176.820,7.946,148.612
C06236=1171.802,300.336,-71.165,-176.817,7.949,148.612
C06237=1171.797,300.584,-71.196,-176.815,7.952,148.612
C06238=1171.793,300.833,-71.225,-176.812,7.955,148.612
C06239=1171.789,301.081,-71.256,-176.810,7.958,148.612
C06240=1171.785,301.329,-71.286,-176.807,7.961,148.612
C06241=1171.780,301.577,-71.316,-176.804,7.964,148.612
C06242=1171.776,301.825,-71.347,-176.802,7.966,148.612
C06243=1171.772,302.073,-71.377,-176.800,7.969,148.612
C06244=1171.768,302.321,-71.408,-176.797,7.972,148.612
C06245=1171.764,302.569,-71.439,-176.795,7.976,148.612
C06246=1171.759,302.818,-71.469,-176.792,7.979,148.612
C06247=1171.755,303.066,-71.499,-176.789,7.982,148.612
C06248=1171.750,303.313,-71.530,-176.787,7.985,148.613
C06249=1171.746,303.562,-71.561,-176.784,7.988,148.613
C06250=1171.743,303.810,-71.591,-176.782,7.991,148.612
C06251=1171.738,304.058,-71.622,-176.779,7.994,148.613
C06252=1171.734,304.305,-71.652,-176.777,7.997,148.613
C06253=1171.730,304.555,-71.682,-176.774,8.000,148.613
C06254=1171.725,304.803,-71.713,-176.771,8.003,148.613
C06255=1171.721,305.050,-71.743,-176.769,8.006,148.613
C06256=1171.717,305.298,-71.774,-176.766,8.010,148.613
C06257=1171.713,305.547,-71.805,-176.764,8.013,148.613
C06258=1171.708,305.795,-71.836,-176.761,8.016,148.613
C06259=1171.704,306.043,-71.866,-176.759,8.019,148.613
C06260=1171.700,306.291,-71.897,-176.756,8.022,148.613
C06261=1171.696,306.539,-71.928,-176.753,8.025,148.613
C06262=1171.692,306.787,-71.958,-176.751,8.028,148.613
C06263=1171.687,307.035,-71.989,-176.748,8.031,148.613
C06264=1171.683,307.283,-72.020,-176.746,8.034,148.613
C06265=1171.678,307.531,-72.051,-176.743,8.037,148.613
C06266=1171.675,307.778,-72.082,-176.740,8.040,148.613
C06267=1171.671,308.027,-72.113,-176.738,8.044,148.614
C06268=1171.666,308.275,-72.144,-176.735,8.047,148.614
C06269=1171.662,308.523,-72.174,-176.733,8.050,148.614
C06270=1171.658,308.772,-72.205,-176.730,8.053,148.614
C06271=1171.654,309.019,-72.236,-176.728,8.056,148.614
C06272=1171.649,309.267,-72.266,-176.725,8.059,148.614
C06273=1171.645,309.516,-72.298,-176.723,8.062,148.614
C06274=1171.641,309.763,-72.329,-176.720,8.066,148.614
C06275=1171.637,310.012,-72.360,-176.718,8.069,148.614
C06276=1171.632,310.260,-72.391,-176.715,8.072,148.614
C06277=1171.628,310.507,-72.421,-176.713,8.075,148.614
C06278=1171.625,310.756,-72.453,-176.710,8.078,148.614
C06279=1171.620,311.003,-72.484,-176.708,8.081,148.614
C06280=1171.615,311.251,-72.514,-176.705,8.084,148.614
C06281=1171.611,311.500,-72.546,-176.703,8.087,148.615
C06282=1171.607,311.747,-72.577,-176.700,8.090,148.615
C06283=1171.603,311.996,-72.608,-176.698,8.094,148.615
C06284=1171.598,312.244,-72.639,-176.695,8.097,148.615
C06285=1171.595,312.492,-72.671,-176.692,8.100,148.615
C06286=1171.590,312.740,-72.702,-176.690,8.103,148.615
C06287=1171.586,312.988,-72.732,-176.687,8.106,148.615
C06288=1171.582,313.236,-72.764,-176.685,8.109,148.615
C06289=1171.578,313.484,-72.794,-176.682,8.112,148.615
C06290=1171.573,313.761,-72.830,-176.679,8.116,148.615
C06291=1171.568,314.037,-72.865,-176.677,8.119,148.615
C06292=1171.564,314.315,-72.899,-176.673,8.123,148.615
C06293=1171.559,314.592,-72.934,-176.671,8.126,148.616
C06294=1171.555,314.839,-72.966,-176.668,8.129,148.616
C06295=1171.551,315.088,-72.997,-176.666,8.133,148.616
C06296=1171.547,315.335,-73.028,-176.663,8.136,148.616
C06297=1171.543,315.584,-73.060,-176.660,8.140,148.616
C06298=1171.538,315.831,-73.091,-176.658,8.143,148.616
C06299=1171.534,316.080,-73.122,-176.655,8.146,148.616
C06300=1171.530,316.327,-73.154,-176.653,8.149,148.616
C06301=1171.526,316.576,-73.185,-176.650,8.152,148.616
C06302=1171.522,316.823,-73.216,-176.648,8.155,148.616
C06303=1171.518,317.072,-73.247,-176.645,8.159,148.616
C06304=1171.513,317.319,-73.279,-176.643,8.162,148.616
C06305=1171.510,317.567,-73.311,-176.640,8.165,148.617
C06306=1171.504,317.816,-73.342,-176.638,8.168,148.617
C06307=1171.501,318.064,-73.374,-176.635,8.171,148.617
C06308=1171.496,318.311,-73.405,-176.633,8.174,148.617
C06309=1171.492,318.560,-73.437,-176.630,8.177,148.617
C06310=1171.489,318.808,-73.468,-176.628,8.180,148.617
C06311=1171.484,319.055,-73.500,-176.625,8.184,148.617
C06312=1171.480,319.304,-73.531,-176.623,8.187,148.617
C06313=1171.475,319.551,-73.563,-176.620,8.190,148.617
C06314=1171.471,319.799,-73.595,-176.618,8.193,148.617
C06315=1171.467,320.047,-73.626,-176.615,8.196,148.618
C06316=1171.463,320.295,-73.658,-176.613,8.200,148.618
C06317=1171.459,320.543,-73.689,-176.610,8.203,148.618
C06318=1171.455,320.791,-73.721,-176.607,8.207,148.618
C06319=1171.451,321.039,-73.753,-176.605,8.210,148.618
C06320=1171.446,321.286,-73.785,-176.602,8.213,148.618
C06321=1171.442,321.535,-73.816,-176.600,8.216,148.618
C06322=1171.439,321.783,-73.848,-176.597,8.219,148.618
C06323=1171.434,322.031,-73.880,-176.595,8.222,148.618
C06324=1171.430,322.279,-73.912,-176.592,8.226,148.619
C06325=1171.426,322.527,-73.944,-176.590,8.229,148.619
C06326=1171.422,322.774,-73.975,-176.587,8.232,148.619
C06327=1171.417,323.023,-74.007,-176.585,8.235,148.619
C06328=1171.414,323.271,-74.039,-176.582,8.238,148.619
C06329=1171.409,323.518,-74.071,-176.580,8.241,148.619
C06330=1171.405,323.767,-74.102,-176.578,8.245,148.619
C06331=1171.401,324.015,-74.134,-176.574,8.249,148.619
C06332=1171.397,324.262,-74.166,-176.572,8.252,148.620
C06333=1171.393,324.510,-74.198,-176.569,8.255,148.620
C06334=1171.389,324.759,-74.230,-176.567,8.258,148.620
C06335=1171.384,325.006,-74.262,-176.565,8.261,148.620
C06336=1171.381,325.253,-74.294,-176.562,8.264,148.620
C06337=1171.376,325.502,-74.327,-176.560,8.268,148.620
C06338=1171.372,325.749,-74.358,-176.557,8.271,148.620
C06339=1171.368,325.997,-74.390,-176.555,8.274,148.620
C06340=1171.364,326.245,-74.422,-176.553,8.277,148.621
C06341=1171.360,326.494,-74.454,-176.550,8.280,148.621
C06342=1171.355,326.741,-74.486,-176.548,8.284,148.621
C06343=1171.351,326.989,-74.518,-176.545,8.288,148.621
C06344=1171.347,327.238,-74.551,-176.542,8.291,148.621
C06345=1171.343,327.486,-74.582,-176.540,8.294,148.621
C06346=1171.339,327.733,-74.615,-176.537,8.297,148.621
C06347=1171.335,327.981,-74.647,-176.535,8.300,148.621
C06348=1171.331,328.229,-74.679,-176.532,8.304,148.622
C06349=1171.327,328.477,-74.711,-176.530,8.307,148.622
C06350=1171.322,328.724,-74.743,-176.527,8.310,148.622
C06351=1171.318,328.972,-74.776,-176.525,8.313,148.622
C06352=1171.315,329.220,-74.808,-176.523,8.316,148.622
C06353=1171.310,329.469,-74.840,-176.520,8.320,148.622
C06354=1171.306,329.716,-74.872,-176.517,8.324,148.622
C06355=1171.302,329.964,-74.905,-176.515,8.327,148.623
C06356=1171.298,330.212,-74.937,-176.512,8.330,148.623
C06357=1171.294,330.460,-74.969,-176.510,8.333,148.623
C06358=1171.289,330.708,-75.002,-176.508,8.336,148.623
C06359=1171.285,330.955,-75.034,-176.505,8.340,148.623
C06360=1171.281,331.203,-75.066,-176.503,8.343,148.623
C06361=1171.277,331.451,-75.099,-176.500,8.347,148.624
C06362=1171.273,331.699,-75.131,-176.498,8.350,148.624
C06363=1171.269,331.947,-75.164,-176.495,8.353,148.624
C06364=1171.265,332.195,-75.196,-176.493,8.356,148.624
C06365=1171.260,332.443,-75.228,-176.490,8.360,148.624
C06366=1171.256,332.690,-75.261,-176.488,8.363,148.624
C06367=1171.252,332.938,-75.293,-176.485,8.366,148.624
C06368=1171.248,333.186,-75.326,-176.483,8.369,148.625
C06369=1171.244,333.434,-75.358,-176.480,8.373,148.625
C06370=1171.240,333.682,-75.391,-176.478,8.377,148.625
C06371=1171.236,333.930,-75.424,-176.475,8.380,148.625
C06372=1171.232,334.177,-75.456,-176.473,8.383,148.625
C06373=1171.227,334.425,-75.489,-176.471,8.386,148.625
C06374=1171.223,334.673,-75.522,-176.468,8.390,148.626
C06375=1171.219,334.921,-75.554,-176.466,8.393,148.626
C06376=1171.215,335.169,-75.587,-176.463,8.396,148.626
C06377=1171.211,335.416,-75.620,-176.460,8.400,148.626
C06378=1171.207,335.665,-75.652,-176.458,8.403,148.626
C06379=1171.203,335.912,-75.685,-176.456,8.407,148.627
C06380=1171.199,336.161,-75.717,-176.453,8.410,148.627
C06381=1171.195,336.408,-75.750,-176.451,8.413,148.627
C06382=1171.191,336.655,-75.783,-176.449,8.416,148.627
C06383=1171.186,336.903,-75.815,-176.446,8.420,148.627
C06384=1171.182,337.151,-75.848,-176.443,8.424,148.627
C06385=1171.178,337.399,-75.881,-176.441,8.427,148.627
C06386=1171.175,337.646,-75.914,-176.438,8.430,148.628
C06387=1171.170,337.895,-75.946,-176.436,8.433,148.628
C06388=1171.166,338.142,-75.980,-176.434,8.437,148.628
C06389=1171.162,338.390,-76.013,-176.432,8.440,148.628
C06390=1171.158,338.638,-76.046,-176.429,8.444,148.628
C06391=1171.154,338.886,-76.078,-176.426,8.447,148.629
C06392=1171.150,339.134,-76.111,-176.424,8.450,148.629
C06393=1171.146,339.381,-76.144,-176.421,8.454,148.629
C06394=1171.141,339.661,-76.182,-176.419,8.458,148.629
C06395=1171.136,339.940,-76.219,-176.416,8.461,148.629
C06396=1171.132,340.219,-76.256,-176.413,8.465,148.630
C06397=1171.127,340.499,-76.292,-176.411,8.469,148.630
C06398=1171.123,340.747,-76.326,-176.408,8.473,148.630
C06399=1171.119,340.995,-76.359,-176.406,8.476,148.630
C06400=1171.115,341.242,-76.392,-176.403,8.479,148.630
C06401=1171.111,341.490,-76.425,-176.400,8.483,148.631
C06402=1171.106,341.738,-76.458,-176.398,8.486,148.631
C06403=1171.102,341.986,-76.491,-176.396,8.490,148.631
C06404=1171.098,342.233,-76.525,-176.394,8.493,148.631
C06405=1171.094,342.481,-76.558,-176.391,8.496,148.631
C06406=1171.090,342.729,-76.591,-176.389,8.499,148.632
C06407=1171.086,342.977,-76.624,-176.386,8.504,148.632
C06408=1171.082,343.224,-76.657,-176.384,8.507,148.632
C06409=1171.077,343.472,-76.690,-176.382,8.510,148.632
C06410=1171.073,343.720,-76.723,-176.379,8.514,148.633
C06411=1171.069,343.967,-76.757,-176.377,8.517,148.633
C06412=1171.065,344.215,-76.790,-176.374,8.521,148.633
C06413=1171.062,344.464,-76.823,-176.372,8.524,148.633
C06414=1171.057,344.711,-76.856,-176.370,8.528,148.633
C06415=1171.053,344.959,-76.890,-176.367,8.531,148.634
C06416=1171.049,345.206,-76.924,-176.365,8.534,148.634
C06417=1171.045,345.454,-76.957,-176.362,8.538,148.634
C06418=1171.041,345.702,-76.990,-176.360,8.542,148.634
C06419=1171.037,345.949,-77.023,-176.358,8.545,148.635
C06420=1171.033,346.197,-77.056,-176.355,8.548,148.635
C06421=1171.029,346.445,-77.089,-176.353,8.551,148.635
C06422=1171.025,346.693,-77.124,-176.350,8.556,148.635
C06423=1171.021,346.940,-77.157,-176.348,8.559,148.635
C06424=1171.016,347.188,-77.190,-176.346,8.562,148.636
C06425=1171.012,347.436,-77.224,-176.343,8.565,148.636
C06426=1171.008,347.683,-77.257,-176.341,8.569,148.636
C06427=1171.004,347.931,-77.291,-176.338,8.573,148.636
C06428=1171.000,348.179,-77.324,-176.336,8.576,148.637
C06429=1170.997,348.427,-77.357,-176.334,8.580,148.637
C06430=1170.992,348.675,-77.392,-176.331,8.583,148.637
C06431=1170.988,348.922,-77.425,-176.328,8.587,148.637
C06432=1170.984,349.170,-77.458,-176.326,8.590,148.637
C06433=1170.980,349.417,-77.492,-176.324,8.594,148.638
C06434=1170.976,349.665,-77.525,-176.322,8.597,148.638
C06435=1170.972,349.913,-77.560,-176.320,8.600,148.638
C06436=1170.968,350.161,-77.593,-176.317,8.605,148.639
C06437=1170.964,350.408,-77.626,-176.315,8.608,148.639
C06438=1170.960,350.656,-77.660,-176.312,8.611,148.639
C06439=1170.956,350.904,-77.694,-176.310,8.614,148.639
C06440=1170.952,351.151,-77.728,-176.307,8.619,148.639
C06441=1170.948,351.399,-77.761,-176.305,8.622,148.640
C06442=1170.944,351.646,-77.795,-176.303,8.625,148.640
C06443=1170.939,351.895,-77.829,-176.301,8.629,148.640
C06444=1170.936,352.142,-77.863,-176.298,8.633,148.641
C06445=1170.931,352.390,-77.896,-176.296,8.636,148.641
C06446=1170.928,352.637,-77.930,-176.293,8.640,148.641
C06447=1170.923,352.886,-77.964,-176.291,8.643,148.641
C06448=1170.920,353.133,-77.998,-176.289,8.647,148.642
C06449=1170.915,353.380,-78.031,-176.286,8.651,148.642
C06450=1170.911,353.628,-78.066,-176.284,8.654,148.642
C06451=1170.908,353.876,-78.100,-176.282,8.657,148.642
C06452=1170.903,354.123,-78.133,-176.279,8.661,148.643
C06453=1170.899,354.371,-78.168,-176.277,8.665,148.643
C06454=1170.896,354.619,-78.202,-176.275,8.668,148.643
C06455=1170.891,354.867,-78.236,-176.273,8.671,148.644
C06456=1170.887,355.114,-78.269,-176.270,8.676,148.644
C06457=1170.883,355.361,-78.303,-176.268,8.679,148.644
C06458=1170.879,355.610,-78.337,-176.266,8.683,148.644
C06459=1170.875,355.857,-78.371,-176.263,8.687,148.645
C06460=1170.870,356.104,-78.406,-176.261,8.690,148.645
C06461=1170.867,356.352,-78.440,-176.259,8.694,148.645
C06462=1170.863,356.600,-78.473,-176.256,8.697,148.646
C06463=1170.859,356.848,-78.508,-176.254,8.701,148.646
C06464=1170.855,357.095,-78.542,-176.252,8.705,148.646
C06465=1170.851,357.342,-78.576,-176.249,8.708,148.646
C06466=1170.847,357.591,-78.610,-176.247,8.711,148.647
C06467=1170.843,357.838,-78.644,-176.245,8.716,148.647
C06468=1170.839,358.085,-78.678,-176.242,8.719,148.647
C06469=1170.835,358.333,-78.713,-176.240,8.722,148.648
C06470=1170.831,358.581,-78.747,-176.238,8.727,148.648
C06471=1170.827,358.829,-78.782,-176.235,8.730,148.648
C06472=1170.823,359.076,-78.816,-176.234,8.734,148.649
C06473=1170.819,359.323,-78.850,-176.231,8.738,148.649
C06474=1170.815,359.571,-78.884,-176.228,8.741,148.649
C06475=1170.810,359.819,-78.918,-176.227,8.745,148.650
C06476=1170.807,360.067,-78.952,-176.224,8.748,148.650
C06477=1170.803,360.314,-78.987,-176.222,8.752,148.650
C06478=1170.798,360.562,-79.021,-176.220,8.756,148.651
C06479=1170.795,360.810,-79.055,-176.218,8.759,148.651
C06480=1170.790,361.057,-79.090,-176.215,8.763,148.651
C06481=1170.787,361.305,-79.124,-176.213,8.767,148.652
C06482=1170.783,361.552,-79.159,-176.211,8.770,148.652
C06483=1170.779,361.800,-79.193,-176.209,8.774,148.652
C06484=1170.775,362.047,-79.228,-176.206,8.778,148.653
C06485=1170.771,362.295,-79.263,-176.204,8.782,148.653
C06486=1170.767,362.542,-79.297,-176.202,8.785,148.653
C06487=1170.763,362.790,-79.332,-176.200,8.788,148.654
C06488=1170.759,363.038,-79.366,-176.198,8.793,148.654
C06489=1170.755,363.285,-79.400,-176.195,8.796,148.654
C06490=1170.751,363.533,-79.435,-176.194,8.800,148.655
C06491=1170.747,363.781,-79.470,-176.192,8.803,148.655
C06492=1170.743,364.027,-79.504,-176.189,8.808,148.656
C06493=1170.739,364.276,-79.539,-176.187,8.811,148.656
C06494=1170.735,364.523,-79.573,-176.185,8.815,148.656
C06495=1170.732,364.771,-79.608,-176.183,8.818,148.657
C06496=1170.727,365.018,-79.642,-176.180,8.823,148.657
C06497=1170.723,365.266,-79.678,-176.179,8.826,148.657
C06498=1170.718,365.548,-79.716,-176.176,8.831,148.658
C06499=1170.714,365.830,-79.756,-176.174,8.834,148.658
C06500=1170.709,366.112,-79.796,-176.172,8.839,148.659
C06501=1170.705,366.394,-79.836,-176.170,8.843,148.659
C06502=1170.702,366.642,-79.870,-176.168,8.847,148.660
C06503=1170.697,366.889,-79.905,-176.166,8.850,148.660
C06504=1170.693,367.137,-79.940,-176.163,8.855,148.661
C06505=1170.689,367.384,-79.974,-176.162,8.858,148.661
C06506=1170.685,367.632,-80.010,-176.160,8.862,148.662
C06507=1170.681,367.879,-80.044,-176.158,8.865,148.662
C06508=1170.678,368.127,-80.079,-176.156,8.869,148.662
C06509=1170.673,368.374,-80.114,-176.154,8.873,148.663
C06510=1170.669,368.622,-80.149,-176.152,8.876,148.663
C06511=1170.665,368.870,-80.184,-176.150,8.880,148.664
C06512=1170.661,369.117,-80.219,-176.148,8.884,148.664
C06513=1170.658,369.364,-80.254,-176.146,8.888,148.665
C06514=1170.653,369.612,-80.288,-176.145,8.892,148.665
C06515=1170.650,369.859,-80.324,-176.143,8.895,148.666
C06516=1170.646,370.107,-80.358,-176.141,8.899,148.666
C06517=1170.641,370.354,-80.394,-176.139,8.903,148.667
C06518=1170.637,370.602,-80.428,-176.138,8.907,148.667
C06519=1170.634,370.850,-80.464,-176.136,8.910,148.668
C06520=1170.629,371.097,-80.498,-176.134,8.914,148.668
C06521=1170.626,371.345,-80.534,-176.133,8.918,148.669
C06522=1170.621,371.592,-80.568,-176.131,8.921,148.669
C06523=1170.618,371.839,-80.603,-176.129,8.925,148.669
C06524=1170.614,372.087,-80.638,-176.128,8.929,148.670
C06525=1170.610,372.334,-80.673,-176.126,8.932,148.671
C06526=1170.606,372.582,-80.709,-176.124,8.936,148.671
C06527=1170.602,372.830,-80.744,-176.123,8.940,148.672
C06528=1170.598,373.076,-80.779,-176.121,8.944,148.672
C06529=1170.594,373.324,-80.814,-176.120,8.947,148.673
C06530=1170.590,373.572,-80.849,-176.118,8.951,148.673
C06531=1170.586,373.819,-80.885,-176.117,8.954,148.674
C06532=1170.582,374.067,-80.919,-176.115,8.958,148.674
C06533=1170.578,374.315,-80.955,-176.114,8.962,148.675
C06534=1170.574,374.561,-80.990,-176.112,8.966,148.676
C06535=1170.570,374.809,-81.026,-176.111,8.969,148.676
C06536=1170.566,375.057,-81.060,-176.110,8.973,148.677
C06537=1170.563,375.304,-81.096,-176.108,8.977,148.677
C06538=1170.559,375.551,-81.131,-176.107,8.980,148.678
C06539=1170.555,375.799,-81.167,-176.105,8.984,148.678
C06540=1170.551,376.047,-81.202,-176.104,8.987,148.679
C06541=1170.546,376.294,-81.237,-176.103,8.991,148.679
C06542=1170.542,376.541,-81.273,-176.101,8.995,148.680
C06543=1170.539,376.789,-81.308,-176.100,8.998,148.681
C06544=1170.535,377.037,-81.343,-176.099,9.002,148.681
C06545=1170.530,377.284,-81.378,-176.098,9.006,148.682
C06546=1170.527,377.531,-81.414,-176.097,9.009,148.682
C06547=1170.523,377.779,-81.450,-176.095,9.013,148.683
C06548=1170.519,378.026,-81.485,-176.095,9.016,148.684
C06549=1170.515,378.273,-81.520,-176.093,9.020,148.684
C06550=1170.511,378.521,-81.555,-176.092,9.024,148.685
C06551=1170.507,378.769,-81.591,-176.091,9.027,148.686
C06552=1170.503,379.017,-81.627,-176.089,9.031,148.686
C06553=1170.499,379.263,-81.662,-176.089,9.034,148.687
C06554=1170.495,379.511,-81.698,-176.087,9.038,148.687
C06555=1170.491,379.758,-81.733,-176.087,9.041,148.688
C06556=1170.488,380.006,-81.769,-176.085,9.045,148.689
C06557=1170.484,380.253,-81.804,-176.084,9.048,148.689
C06558=1170.479,380.501,-81.840,-176.084,9.051,148.690
C06559=1170.476,380.748,-81.875,-176.083,9.055,148.691
C06560=1170.472,380.996,-81.911,-176.082,9.059,148.691
C06561=1170.468,381.242,-81.946,-176.081,9.062,148.692
C06562=1170.464,381.490,-81.982,-176.080,9.066,148.693
C06563=1170.460,381.738,-82.018,-176.079,9.069,148.693
C06564=1170.456,381.985,-82.053,-176.078,9.072,148.694
C06565=1170.452,382.233,-82.089,-176.077,9.076,148.695
C06566=1170.448,382.479,-82.124,-176.076,9.079,148.695
C06567=1170.444,382.727,-82.160,-176.076,9.083,148.696
C06568=1170.440,382.975,-82.196,-176.075,9.086,148.697
C06569=1170.436,383.222,-82.231,-176.075,9.089,148.697
C06570=1170.433,383.470,-82.267,-176.073,9.093,148.698
C06571=1170.429,383.717,-82.303,-176.073,9.096,148.699
C06572=1170.424,383.964,-82.338,-176.072,9.100,148.699
C06573=1170.420,384.212,-82.374,-176.072,9.103,148.700
C06574=1170.417,384.459,-82.409,-176.071,9.106,148.701
C06575=1170.413,384.707,-82.445,-176.070,9.109,148.701
C06576=1170.408,384.955,-82.481,-176.070,9.113,148.702
C06577=1170.405,385.202,-82.517,-176.070,9.116,148.703
C06578=1170.401,385.449,-82.552,-176.069,9.119,148.704
C06579=1170.397,385.696,-82.588,-176.068,9.123,148.704
C06580=1170.393,385.944,-82.624,-176.068,9.126,148.705
C06581=1170.389,386.191,-82.660,-176.068,9.128,148.706
C06582=1170.385,386.439,-82.695,-176.067,9.132,148.706
C06583=1170.381,386.686,-82.731,-176.067,9.135,148.707
C06584=1170.377,386.934,-82.767,-176.066,9.139,148.708
C06585=1170.373,387.180,-82.803,-176.066,9.142,148.709
C06586=1170.370,387.428,-82.838,-176.066,9.144,148.709
C06587=1170.365,387.675,-82.875,-176.065,9.148,148.710
C06588=1170.362,387.923,-82.910,-176.065,9.151,148.711
C06589=1170.358,388.170,-82.946,-176.065,9.154,148.712
C06590=1170.354,388.418,-82.982,-176.065,9.157,148.712
C06591=1170.350,388.665,-83.018,-176.064,9.160,148.713
C06592=1170.346,388.912,-83.053,-176.064,9.163,148.714
C06593=1170.342,389.160,-83.089,-176.064,9.166,148.715
C06594=1170.338,389.407,-83.125,-176.064,9.169,148.715
C06595=1170.335,389.654,-83.161,-176.063,9.172,148.716
C06596=1170.330,389.902,-83.197,-176.063,9.175,148.717
C06597=1170.327,390.149,-83.233,-176.063,9.178,148.717
C06598=1170.323,390.397,-83.268,-176.063,9.180,148.718
C06599=1170.319,390.644,-83.305,-176.063,9.184,148.719
C06600=1170.315,390.892,-83.341,-176.063,9.186,148.720
C06601=1170.311,391.139,-83.376,-176.063,9.189,148.720
C06602=1170.307,391.424,-83.417,-176.063,9.193,148.721
C06603=1170.302,391.709,-83.459,-176.063,9.196,148.722
C06604=1170.297,391.994,-83.500,-176.063,9.199,148.723
C06605=1170.293,392.278,-83.542,-176.063,9.202,148.724
C06606=1170.289,392.526,-83.578,-176.063,9.205,148.724
C06607=1170.285,392.773,-83.614,-176.063,9.207,148.725
C06608=1170.281,393.020,-83.650,-176.063,9.211,148.726
C06609=1170.278,393.268,-83.685,-176.063,9.213,148.727
C06610=1170.273,393.516,-83.722,-176.063,9.216,148.727
C06611=1170.270,393.762,-83.758,-176.063,9.219,148.728
C06612=1170.265,394.010,-83.794,-176.063,9.221,148.729
C06613=1170.262,394.258,-83.830,-176.063,9.224,148.729
C06614=1170.258,394.505,-83.866,-176.064,9.226,148.730
C06615=1170.254,394.752,-83.902,-176.064,9.229,148.731
C06616=1170.250,395.000,-83.938,-176.064,9.232,148.732
C06617=1170.246,395.246,-83.974,-176.064,9.234,148.733
C06618=1170.242,395.494,-84.010,-176.065,9.237,148.733
C06619=1170.238,395.742,-84.046,-176.065,9.239,148.734
C06620=1170.234,395.989,-84.082,-176.065,9.242,148.735
C06621=1170.231,396.236,-84.118,-176.065,9.245,148.735
C06622=1170.226,396.484,-84.154,-176.065,9.247,148.736
C06623=1170.223,396.731,-84.190,-176.065,9.250,148.737
C06624=1170.218,396.979,-84.226,-176.065,9.252,148.738
C06625=1170.215,397.225,-84.262,-176.066,9.255,148.738
C06626=1170.211,397.473,-84.298,-176.066,9.257,148.739
C06627=1170.207,397.721,-84.334,-176.066,9.260,148.740
C06628=1170.204,397.968,-84.370,-176.067,9.262,148.740
C06629=1170.199,398.215,-84.406,-176.067,9.264,148.741
C06630=1170.196,398.462,-84.443,-176.067,9.267,148.742
C06631=1170.191,398.710,-84.479,-176.067,9.269,148.742
C06632=1170.187,398.957,-84.514,-176.067,9.272,148.743
C06633=1170.183,399.204,-84.551,-176.068,9.274,148.744
C06634=1170.179,399.452,-84.586,-176.068,9.276,148.745
C06635=1170.175,399.699,-84.623,-176.068,9.279,148.745
C06636=1170.172,399.946,-84.659,-176.068,9.281,148.746
C06637=1170.167,400.194,-84.695,-176.069,9.283,148.746
C06638=1170.164,400.441,-84.731,-176.069,9.285,148.747
C06639=1170.160,400.689,-84.767,-176.069,9.288,148.748
C06640=1170.156,400.936,-84.804,-176.070,9.290,148.749
C06641=1170.152,401.183,-84.839,-176.070,9.292,148.749
C06642=1170.148,401.430,-84.876,-176.070,9.295,148.750
C06643=1170.145,401.678,-84.912,-176.071,9.297,148.751
C06644=1170.140,401.926,-84.948,-176.071,9.299,148.751
C06645=1170.137,402.173,-84.984,-176.072,9.301,148.752
C06646=1170.133,402.420,-85.020,-176.072,9.304,148.753
C06647=1170.129,402.667,-85.056,-176.072,9.306,148.753
C06648=1170.125,402.915,-85.093,-176.072,9.308,148.754
C06649=1170.121,403.162,-85.129,-176.072,9.310,148.755
C06650=1170.117,403.410,-85.165,-176.073,9.312,148.755
C06651=1170.114,403.657,-85.201,-176.073,9.314,148.756
C06652=1170.109,403.905,-85.237,-176.074,9.316,148.757
C06653=1170.106,404.152,-85.273,-176.074,9.319,148.757
C06654=1170.102,404.399,-85.310,-176.074,9.320,148.758
C06655=1170.097,404.646,-85.345,-176.074,9.323,148.758
C06656=1170.093,404.893,-85.382,-176.075,9.324,148.759
C06657=1170.090,405.141,-85.417,-176.075,9.327,148.760
C06658=1170.085,405.388,-85.454,-176.076,9.329,148.760
C06659=1170.082,405.635,-85.490,-176.076,9.331,148.761
C06660=1170.078,405.883,-85.527,-176.076,9.333,148.762
C06661=1170.074,406.130,-85.562,-176.077,9.335,148.762
C06662=1170.070,406.377,-85.599,-176.077,9.337,148.763
C06663=1170.066,406.625,-85.635,-176.078,9.339,148.763
C06664=1170.062,406.872,-85.671,-176.078,9.341,148.764
C06665=1170.058,407.119,-85.707,-176.078,9.343,148.765
C06666=1170.054,407.367,-85.744,-176.078,9.345,148.765
C06667=1170.051,407.614,-85.779,-176.079,9.347,148.766
C06668=1170.047,407.861,-85.816,-176.080,9.349,148.767
C06669=1170.043,408.109,-85.852,-176.079,9.351,148.767
C06670=1170.039,408.356,-85.889,-176.080,9.353,148.768
C06671=1170.035,408.604,-85.924,-176.080,9.355,148.769
C06672=1170.031,408.851,-85.961,-176.080,9.357,148.769
C06673=1170.027,409.098,-85.997,-176.081,9.358,148.770
C06674=1170.023,409.345,-86.033,-176.081,9.361,148.770
C06675=1170.020,409.593,-86.069,-176.082,9.362,148.771
C06676=1170.016,409.840,-86.106,-176.082,9.364,148.771
C06677=1170.012,410.088,-86.141,-176.082,9.366,148.772
C06678=1170.008,410.335,-86.178,-176.083,9.368,148.773
C06679=1170.005,410.582,-86.215,-176.083,9.370,148.773
C06680=1170.000,410.829,-86.251,-176.083,9.372,148.774
C06681=1169.996,411.077,-86.288,-176.084,9.374,148.774
C06682=1169.992,411.324,-86.323,-176.084,9.375,148.775
C06683=1169.988,411.571,-86.360,-176.084,9.378,148.776
C06684=1169.985,411.819,-86.395,-176.085,9.379,148.776
C06685=1169.980,412.066,-86.432,-176.085,9.381,148.777
C06686=1169.977,412.314,-86.468,-176.085,9.383,148.777
C06687=1169.973,412.561,-86.505,-176.086,9.385,148.778
C06688=1169.969,412.808,-86.540,-176.086,9.386,148.778
C06689=1169.965,413.055,-86.577,-176.086,9.389,148.779
C06690=1169.962,413.302,-86.613,-176.086,9.390,148.779
C06691=1169.957,413.550,-86.650,-176.087,9.392,148.780
C06692=1169.953,413.797,-86.686,-176.087,9.394,148.781
C06693=1169.949,414.045,-86.722,-176.088,9.396,148.781
C06694=1169.945,414.292,-86.759,-176.088,9.398,148.782
C06695=1169.942,414.540,-86.794,-176.088,9.399,148.782
C06696=1169.938,414.787,-86.831,-176.088,9.402,148.783
C06697=1169.934,415.034,-86.867,-176.089,9.403,148.783
C06698=1169.930,415.281,-86.904,-176.089,9.405,148.784
C06699=1169.926,415.528,-86.940,-176.090,9.406,148.784
C06700=1169.924,415.776,-86.977,-176.089,9.409,148.785
C06701=1169.922,416.023,-87.012,-176.090,9.410,148.786
C06702=1169.922,416.312,-87.055,-176.090,9.412,148.786
C06703=1169.922,416.599,-87.096,-176.090,9.414,148.787
C06704=1169.925,416.888,-87.138,-176.091,9.416,148.787
C06705=1169.928,417.175,-87.179,-176.091,9.417,148.788
C06706=1169.507,417.176,-87.224,-176.094,9.428,148.791
C06707=1169.503,416.885,-87.181,-176.094,9.427,148.791
C06708=1169.501,416.595,-87.140,-176.093,9.425,148.790
C06709=1169.501,416.304,-87.097,-176.094,9.423,148.790
C06710=1169.501,416.012,-87.055,-176.093,9.421,148.789
C06711=1169.503,415.765,-87.019,-176.093,9.420,148.789
C06712=1169.506,415.517,-86.983,-176.092,9.417,148.788
C06713=1169.509,415.271,-86.946,-176.092,9.416,148.788
C06714=1169.513,415.023,-86.911,-176.092,9.414,148.787
C06715=1169.517,414.776,-86.874,-176.091,9.412,148.786
C06716=1169.521,414.528,-86.838,-176.091,9.410,148.786
C06717=1169.524,414.280,-86.801,-176.091,9.408,148.785
C06718=1169.528,414.033,-86.764,-176.090,9.407,148.785
C06719=1169.532,413.786,-86.729,-176.090,9.405,148.784
C06720=1169.536,413.539,-86.692,-176.090,9.403,148.784
C06721=1169.540,413.291,-86.656,-176.090,9.401,148.783
C06722=1169.544,413.044,-86.620,-176.089,9.400,148.783
C06723=1169.547,412.796,-86.584,-176.089,9.397,148.782
C06724=1169.551,412.549,-86.547,-176.089,9.396,148.781
C06725=1169.556,412.302,-86.510,-176.088,9.394,148.781
C06726=1169.559,412.055,-86.475,-176.088,9.392,148.780
C06727=1169.563,411.807,-86.438,-176.088,9.390,148.780
C06728=1169.567,411.560,-86.402,-176.087,9.389,148.779
C06729=1169.571,411.313,-86.366,-176.087,9.387,148.779
C06730=1169.575,411.065,-86.330,-176.087,9.385,148.778
C06731=1169.579,410.818,-86.293,-176.086,9.383,148.777
C06732=1169.583,410.570,-86.258,-176.086,9.381,148.777
C06733=1169.587,410.323,-86.221,-176.086,9.379,148.776
C06734=1169.590,410.076,-86.185,-176.085,9.377,148.776
C06735=1169.594,409.829,-86.148,-176.085,9.376,148.775
C06736=1169.599,409.582,-86.112,-176.084,9.373,148.774
C06737=1169.603,409.335,-86.076,-176.084,9.372,148.774
C06738=1169.607,409.087,-86.039,-176.083,9.370,148.773
C06739=1169.610,408.840,-86.004,-176.084,9.368,148.773
C06740=1169.615,408.593,-85.967,-176.083,9.366,148.772
C06741=1169.618,408.345,-85.931,-176.082,9.364,148.771
C06742=1169.622,408.098,-85.895,-176.083,9.362,148.771
C06743=1169.626,407.851,-85.859,-176.082,9.360,148.770
C06744=1169.630,407.603,-85.822,-176.082,9.358,148.770
C06745=1169.634,407.356,-85.787,-176.081,9.356,148.769
C06746=1169.638,407.109,-85.750,-176.081,9.354,148.768
C06747=1169.642,406.861,-85.714,-176.081,9.352,148.768
C06748=1169.646,406.614,-85.677,-176.080,9.350,148.767
C06749=1169.649,406.366,-85.642,-176.080,9.348,148.767
C06750=1169.653,406.119,-85.605,-176.079,9.346,148.766
C06751=1169.657,405.872,-85.569,-176.079,9.344,148.765
C06752=1169.661,405.625,-85.533,-176.079,9.342,148.765
C06753=1169.665,405.377,-85.497,-176.078,9.340,148.764
C06754=1169.669,405.130,-85.460,-176.078,9.338,148.763
C06755=1169.673,404.882,-85.425,-176.077,9.336,148.763
C06756=1169.677,404.635,-85.388,-176.077,9.333,148.762
C06757=1169.680,404.388,-85.352,-176.077,9.332,148.761
C06758=1169.684,404.141,-85.315,-176.077,9.329,148.761
C06759=1169.688,403.893,-85.280,-176.076,9.328,148.760
C06760=1169.692,403.646,-85.243,-176.076,9.325,148.760
C06761=1169.696,403.398,-85.207,-176.075,9.323,148.759
C06762=1169.700,403.151,-85.171,-176.075,9.321,148.758
C06763=1169.704,402.904,-85.135,-176.074,9.319,148.757
C06764=1169.708,402.656,-85.098,-176.074,9.316,148.757
C06765=1169.711,402.409,-85.063,-176.074,9.315,148.756
C06766=1169.715,402.162,-85.026,-176.074,9.312,148.756
C06767=1169.719,401.914,-84.990,-176.074,9.310,148.755
C06768=1169.723,401.666,-84.954,-176.073,9.308,148.754
C06769=1169.727,401.420,-84.918,-176.073,9.306,148.754
C06770=1169.731,401.172,-84.882,-176.072,9.304,148.753
C06771=1169.735,400.925,-84.845,-176.072,9.301,148.752
C06772=1169.739,400.677,-84.809,-176.072,9.299,148.751
C06773=1169.742,400.430,-84.773,-176.071,9.297,148.751
C06774=1169.747,400.182,-84.737,-176.071,9.294,148.750
C06775=1169.750,399.935,-84.701,-176.071,9.292,148.749
C06776=1169.755,399.688,-84.664,-176.070,9.290,148.749
C06777=1169.759,399.441,-84.629,-176.070,9.288,148.748
C06778=1169.763,399.194,-84.592,-176.070,9.285,148.747
C06779=1169.767,398.946,-84.557,-176.070,9.282,148.747
C06780=1169.770,398.699,-84.521,-176.069,9.281,148.746
C06781=1169.774,398.451,-84.484,-176.069,9.278,148.745
C06782=1169.778,398.204,-84.449,-176.069,9.275,148.744
C06783=1169.782,397.957,-84.412,-176.069,9.273,148.744
C06784=1169.786,397.709,-84.376,-176.068,9.270,148.743
C06785=1169.790,397.462,-84.340,-176.068,9.269,148.742
C06786=1169.793,397.215,-84.304,-176.068,9.266,148.742
C06787=1169.798,396.967,-84.268,-176.067,9.263,148.741
C06788=1169.801,396.720,-84.232,-176.067,9.261,148.740
C06789=1169.805,396.472,-84.196,-176.067,9.258,148.740
C06790=1169.809,396.225,-84.159,-176.067,9.256,148.739
C06791=1169.813,395.978,-84.124,-176.067,9.253,148.738
C06792=1169.817,395.730,-84.088,-176.067,9.251,148.737
C06793=1169.821,395.484,-84.052,-176.066,9.248,148.737
C06794=1169.825,395.236,-84.016,-176.066,9.245,148.736
C06795=1169.829,394.988,-83.980,-176.066,9.243,148.735
C06796=1169.833,394.741,-83.943,-176.066,9.240,148.735
C06797=1169.837,394.494,-83.908,-176.066,9.238,148.734
C06798=1169.840,394.246,-83.872,-176.066,9.235,148.733
C06799=1169.845,393.999,-83.835,-176.066,9.233,148.732
C06800=1169.848,393.752,-83.800,-176.065,9.230,148.732
C06801=1169.853,393.504,-83.763,-176.065,9.227,148.731
C06802=1169.856,393.257,-83.727,-176.065,9.225,148.730
C06803=1169.860,393.009,-83.692,-176.065,9.222,148.729
C06804=1169.864,392.762,-83.656,-176.065,9.219,148.729
C06805=1169.867,392.515,-83.619,-176.065,9.216,148.728
C06806=1169.872,392.268,-83.583,-176.065,9.214,148.727
C06807=1169.876,391.983,-83.542,-176.065,9.210,148.726
C06808=1169.881,391.698,-83.501,-176.065,9.207,148.725
C06809=1169.885,391.413,-83.460,-176.065,9.204,148.725
C06810=1169.889,391.128,-83.418,-176.065,9.200,148.724
C06811=1169.894,390.881,-83.383,-176.065,9.198,148.723
C06812=1169.898,390.633,-83.346,-176.065,9.195,148.722
C06813=1169.901,390.386,-83.310,-176.065,9.192,148.722
C06814=1169.906,390.138,-83.274,-176.065,9.189,148.721
C06815=1169.909,389.891,-83.239,-176.065,9.186,148.720
C06816=1169.913,389.643,-83.203,-176.065,9.183,148.719
C06817=1169.917,389.396,-83.166,-176.066,9.180,148.719
C06818=1169.921,389.149,-83.131,-176.065,9.177,148.718
C06819=1169.925,388.901,-83.095,-176.066,9.174,148.717
C06820=1169.929,388.653,-83.059,-176.066,9.172,148.717
C06821=1169.933,388.407,-83.023,-176.067,9.168,148.716
C06822=1169.937,388.160,-82.987,-176.066,9.166,148.715
C06823=1169.941,387.912,-82.951,-176.067,9.162,148.714
C06824=1169.945,387.664,-82.916,-176.067,9.159,148.714
C06825=1169.948,387.417,-82.880,-176.067,9.156,148.713
C06826=1169.952,387.170,-82.843,-176.067,9.153,148.712
C06827=1169.956,386.922,-82.808,-176.068,9.149,148.711
C06828=1169.960,386.675,-82.772,-176.069,9.146,148.711
C06829=1169.964,386.428,-82.737,-176.069,9.143,148.710
C06830=1169.968,386.180,-82.701,-176.069,9.140,148.709
C06831=1169.972,385.932,-82.665,-176.069,9.137,148.708
C06832=1169.975,385.686,-82.629,-176.070,9.134,148.708
C06833=1169.980,385.438,-82.593,-176.071,9.131,148.707
C06834=1169.983,385.190,-82.557,-176.071,9.127,148.706
C06835=1169.987,384.943,-82.522,-176.072,9.124,148.706
C06836=1169.991,384.696,-82.487,-176.072,9.121,148.705
C06837=1169.996,384.448,-82.451,-176.073,9.117,148.704
C06838=1169.999,384.201,-82.415,-176.073,9.114,148.703
C06839=1170.003,383.953,-82.379,-176.074,9.111,148.703
C06840=1170.007,383.706,-82.343,-176.074,9.107,148.702
C06841=1170.011,383.458,-82.307,-176.075,9.104,148.702
C06842=1170.015,383.212,-82.272,-176.076,9.100,148.701
C06843=1170.019,382.964,-82.236,-176.077,9.097,148.700
C06844=1170.022,382.717,-82.201,-176.078,9.094,148.699
C06845=1170.027,382.469,-82.165,-176.078,9.091,148.699
C06846=1170.030,382.221,-82.129,-176.079,9.087,148.698
C06847=1170.035,381.975,-82.094,-176.080,9.083,148.697
C06848=1170.038,381.727,-82.058,-176.081,9.080,148.697
C06849=1170.043,381.479,-82.022,-176.082,9.077,148.696
C06850=1170.046,381.232,-81.987,-176.083,9.073,148.695
C06851=1170.050,380.984,-81.951,-176.083,9.069,148.695
C06852=1170.054,380.737,-81.916,-176.084,9.066,148.694
C06853=1170.058,380.490,-81.880,-176.086,9.062,148.693
C06854=1170.062,380.242,-81.844,-176.086,9.059,148.693
C06855=1170.066,379.995,-81.809,-176.087,9.056,148.692
C06856=1170.070,379.747,-81.773,-176.088,9.052,148.691
C06857=1170.074,379.500,-81.738,-176.089,9.049,148.691
C06858=1170.078,379.253,-81.702,-176.090,9.045,148.690
C06859=1170.082,379.005,-81.668,-176.091,9.042,148.689
C06860=1170.085,378.757,-81.632,-176.092,9.038,148.689
C06861=1170.090,378.510,-81.596,-176.093,9.035,148.688
C06862=1170.094,378.263,-81.561,-176.095,9.031,148.688
C06863=1170.098,378.015,-81.525,-176.096,9.027,148.687
C06864=1170.101,377.768,-81.490,-176.097,9.024,148.686
C06865=1170.106,377.521,-81.454,-176.098,9.020,148.686
C06866=1170.109,377.273,-81.419,-176.099,9.017,148.685
C06867=1170.113,377.025,-81.384,-176.101,9.013,148.685
C06868=1170.117,376.778,-81.348,-176.102,9.009,148.684
C06869=1170.122,376.531,-81.313,-176.103,9.006,148.683
C06870=1170.126,376.283,-81.277,-176.104,9.002,148.683
C06871=1170.129,376.036,-81.242,-176.106,8.998,148.682
C06872=1170.133,375.787,-81.207,-176.107,8.994,148.681
C06873=1170.137,375.541,-81.172,-176.108,8.991,148.681
C06874=1170.141,375.293,-81.136,-176.110,8.987,148.680
C06875=1170.145,375.046,-81.101,-176.111,8.984,148.680
C06876=1170.149,374.798,-81.066,-176.113,8.980,148.679
C06877=1170.153,374.551,-81.030,-176.114,8.976,148.679
C06878=1170.157,374.303,-80.995,-176.115,8.973,148.678
C06879=1170.161,374.056,-80.960,-176.117,8.969,148.678
C06880=1170.165,373.808,-80.925,-176.119,8.965,148.677
C06881=1170.169,373.561,-80.889,-176.120,8.961,148.677
C06882=1170.173,373.313,-80.855,-176.122,8.958,148.676
C06883=1170.177,373.066,-80.819,-176.123,8.954,148.675
C06884=1170.180,372.818,-80.784,-176.125,8.950,148.675
C06885=1170.184,372.570,-80.749,-176.127,8.946,148.674
C06886=1170.189,372.323,-80.714,-176.128,8.943,148.674
C06887=1170.192,372.076,-80.678,-176.130,8.939,148.673
C06888=1170.196,371.828,-80.643,-176.132,8.935,148.673
C06889=1170.201,371.581,-80.608,-176.133,8.931,148.672
C06890=1170.205,371.333,-80.573,-176.135,8.928,148.672
C06891=1170.209,371.086,-80.538,-176.136,8.924,148.671
C06892=1170.212,370.839,-80.503,-176.138,8.920,148.671
C06893=1170.216,370.591,-80.468,-176.140,8.917,148.670
C06894=1170.220,370.344,-80.433,-176.142,8.913,148.670
C06895=1170.224,370.096,-80.398,-176.143,8.909,148.669
C06896=1170.228,369.848,-80.363,-176.145,8.906,148.669
C06897=1170.232,369.601,-80.328,-176.147,8.902,148.668
C06898=1170.236,369.354,-80.293,-176.149,8.898,148.668
C06899=1170.240,369.106,-80.258,-176.151,8.895,148.668
C06900=1170.244,368.858,-80.224,-176.152,8.891,148.667
C06901=1170.247,368.611,-80.189,-176.154,8.887,148.667
C06902=1170.252,368.363,-80.154,-176.156,8.884,148.666
C06903=1170.256,368.116,-80.119,-176.158,8.880,148.666
C06904=1170.260,367.868,-80.084,-176.160,8.876,148.665
C06905=1170.264,367.620,-80.049,-176.162,8.872,148.665
C06906=1170.268,367.374,-80.014,-176.164,8.868,148.664
C06907=1170.272,367.126,-79.980,-176.166,8.865,148.664
C06908=1170.275,366.878,-79.944,-176.167,8.861,148.664
C06909=1170.280,366.631,-79.910,-176.169,8.858,148.663
C06910=1170.284,366.383,-79.875,-176.172,8.853,148.663
C06911=1170.289,366.101,-79.836,-176.174,8.850,148.662
C06912=1170.293,365.819,-79.796,-176.176,8.845,148.662
C06913=1170.297,365.536,-79.756,-176.178,8.841,148.661
C06914=1170.302,365.255,-79.716,-176.181,8.837,148.661
C06915=1170.305,365.007,-79.682,-176.183,8.833,148.661
C06916=1170.310,364.759,-79.648,-176.185,8.829,148.660
C06917=1170.314,364.512,-79.612,-176.187,8.825,148.660
C06918=1170.318,364.265,-79.578,-176.190,8.822,148.659
C06919=1170.321,364.017,-79.544,-176.191,8.818,148.659
C06920=1170.326,363.769,-79.509,-176.193,8.814,148.659
C06921=1170.330,363.521,-79.474,-176.196,8.810,148.658
C06922=1170.334,363.274,-79.440,-176.198,8.807,148.658
C06923=1170.337,363.027,-79.405,-176.200,8.803,148.657
C06924=1170.342,362.779,-79.370,-176.202,8.800,148.657
C06925=1170.345,362.531,-79.336,-176.205,8.795,148.657
C06926=1170.350,362.284,-79.302,-176.206,8.792,148.656
C06927=1170.353,362.036,-79.267,-176.209,8.788,148.656
C06928=1170.358,361.789,-79.233,-176.211,8.784,148.656
C06929=1170.362,361.541,-79.198,-176.213,8.781,148.655
C06930=1170.365,361.293,-79.164,-176.215,8.777,148.655
C06931=1170.369,361.045,-79.129,-176.218,8.774,148.655
C06932=1170.374,360.798,-79.095,-176.220,8.769,148.654
C06933=1170.378,360.551,-79.061,-176.222,8.766,148.654
C06934=1170.382,360.303,-79.026,-176.224,8.762,148.654
C06935=1170.386,360.056,-78.992,-176.227,8.758,148.653
C06936=1170.389,359.807,-78.958,-176.229,8.755,148.653
C06937=1170.393,359.560,-78.924,-176.231,8.751,148.653
C06938=1170.397,359.312,-78.889,-176.234,8.747,148.652
C06939=1170.401,359.065,-78.855,-176.236,8.744,148.652
C06940=1170.406,358.818,-78.821,-176.238,8.740,148.652
C06941=1170.409,358.570,-78.786,-176.240,8.737,148.651
C06942=1170.413,358.322,-78.752,-176.243,8.733,148.651
C06943=1170.417,358.075,-78.718,-176.245,8.729,148.651
C06944=1170.422,357.827,-78.684,-176.247,8.726,148.650
C06945=1170.425,357.580,-78.650,-176.250,8.722,148.650
C06946=1170.429,357.331,-78.615,-176.252,8.718,148.650
C06947=1170.433,357.084,-78.581,-176.254,8.715,148.649
C06948=1170.438,356.837,-78.547,-176.256,8.711,148.649
C06949=1170.441,356.589,-78.513,-176.259,8.707,148.649
C06950=1170.446,356.341,-78.479,-176.261,8.704,148.649
C06951=1170.450,356.094,-78.445,-176.263,8.700,148.648
C06952=1170.454,355.846,-78.410,-176.266,8.696,148.648
C06953=1170.458,355.599,-78.376,-176.268,8.693,148.648
C06954=1170.462,355.351,-78.343,-176.270,8.689,148.647
C06955=1170.466,355.103,-78.308,-176.272,8.686,148.647
C06956=1170.469,354.856,-78.274,-176.275,8.682,148.647
C06957=1170.474,354.608,-78.241,-176.278,8.679,148.647
C06958=1170.478,354.360,-78.206,-176.279,8.675,148.646
C06959=1170.481,354.113,-78.172,-176.282,8.671,148.646
C06960=1170.486,353.865,-78.139,-176.285,8.668,148.646
C06961=1170.490,353.617,-78.104,-176.287,8.664,148.646
C06962=1170.494,353.369,-78.071,-176.289,8.661,148.645
C06963=1170.498,353.122,-78.037,-176.292,8.657,148.645
C06964=1170.502,352.875,-78.003,-176.294,8.653,148.645
C06965=1170.506,352.626,-77.969,-176.296,8.650,148.644
C06966=1170.510,352.379,-77.935,-176.298,8.647,148.644
C06967=1170.514,352.131,-77.902,-176.301,8.642,148.644
C06968=1170.518,351.883,-77.868,-176.303,8.639,148.644
C06969=1170.522,351.635,-77.834,-176.305,8.636,148.643
C06970=1170.526,351.388,-77.800,-176.308,8.632,148.643
C06971=1170.530,351.140,-77.767,-176.310,8.628,148.643
C06972=1170.534,350.893,-77.733,-176.313,8.625,148.643
C06973=1170.539,350.645,-77.699,-176.315,8.622,148.642
C06974=1170.542,350.397,-77.665,-176.317,8.618,148.642
C06975=1170.546,350.150,-77.632,-176.320,8.614,148.642
C06976=1170.550,349.903,-77.598,-176.322,8.611,148.642
C06977=1170.555,349.654,-77.564,-176.324,8.607,148.641
C06978=1170.559,349.406,-77.531,-176.327,8.604,148.641
C06979=1170.563,349.159,-77.497,-176.329,8.600,148.641
C06980=1170.567,348.911,-77.464,-176.332,8.597,148.641
C06981=1170.571,348.664,-77.431,-176.334,8.593,148.640
C06982=1170.575,348.415,-77.396,-176.336,8.590,148.640
C06983=1170.579,348.168,-77.363,-176.339,8.587,148.640
C06984=1170.583,347.920,-77.329,-176.341,8.583,148.640
C06985=1170.587,347.673,-77.295,-176.343,8.579,148.639
C06986=1170.591,347.425,-77.262,-176.346,8.576,148.639
C06987=1170.595,347.177,-77.229,-176.348,8.572,148.639
C06988=1170.599,346.930,-77.196,-176.351,8.568,148.639
C06989=1170.603,346.682,-77.161,-176.353,8.565,148.638
C06990=1170.607,346.434,-77.128,-176.355,8.562,148.638
C06991=1170.612,346.186,-77.095,-176.358,8.558,148.638
C06992=1170.616,345.938,-77.062,-176.360,8.555,148.638
C06993=1170.620,345.691,-77.029,-176.363,8.551,148.638
C06994=1170.624,345.444,-76.995,-176.365,8.548,148.637
C06995=1170.628,345.196,-76.962,-176.367,8.544,148.637
C06996=1170.632,344.948,-76.928,-176.370,8.541,148.637
C06997=1170.635,344.700,-76.895,-176.372,8.538,148.637
C06998=1170.640,344.452,-76.862,-176.375,8.534,148.636
C06999=1170.644,344.204,-76.829,-176.377,8.530,148.636
C07000=1170.648,343.956,-76.795,-176.379,8.527,148.636
C07001=1170.652,343.709,-76.762,-176.382,8.524,148.636
C07002=1170.656,343.461,-76.729,-176.384,8.520,148.636
C07003=1170.660,343.213,-76.696,-176.387,8.516,148.635
C07004=1170.664,342.966,-76.663,-176.389,8.513,148.635
C07005=1170.668,342.718,-76.629,-176.391,8.510,148.635
C07006=1170.672,342.471,-76.596,-176.394,8.507,148.635
C07007=1170.677,342.222,-76.563,-176.396,8.503,148.635
C07008=1170.681,341.975,-76.530,-176.399,8.499,148.634
C07009=1170.685,341.727,-76.497,-176.401,8.496,148.634
C07010=1170.689,341.479,-76.464,-176.404,8.493,148.634
C07011=1170.693,341.231,-76.431,-176.406,8.489,148.634
C07012=1170.698,340.984,-76.398,-176.408,8.486,148.634
C07013=1170.702,340.736,-76.364,-176.411,8.482,148.633
C07014=1170.706,340.488,-76.331,-176.413,8.479,148.633
C07015=1170.710,340.209,-76.294,-176.416,8.475,148.633
C07016=1170.715,339.929,-76.256,-176.419,8.471,148.633
C07017=1170.719,339.651,-76.220,-176.422,8.467,148.633
C07018=1170.724,339.371,-76.182,-176.425,8.463,148.632
C07019=1170.729,339.123,-76.150,-176.427,8.460,148.632
C07020=1170.733,338.875,-76.116,-176.429,8.457,148.632
C07021=1170.737,338.627,-76.083,-176.432,8.453,148.632
C07022=1170.740,338.380,-76.051,-176.434,8.450,148.631
C07023=1170.745,338.131,-76.018,-176.436,8.447,148.631
C07024=1170.749,337.884,-75.985,-176.439,8.443,148.631
C07025=1170.753,337.636,-75.952,-176.442,8.440,148.631
C07026=1170.757,337.388,-75.919,-176.444,8.436,148.631
C07027=1170.761,337.140,-75.887,-176.446,8.433,148.631
C07028=1170.765,336.892,-75.854,-176.449,8.430,148.630
C07029=1170.769,336.645,-75.821,-176.451,8.426,148.630
C07030=1170.773,336.396,-75.788,-176.454,8.423,148.630
C07031=1170.777,336.149,-75.756,-176.456,8.419,148.630
C07032=1170.781,335.901,-75.723,-176.459,8.416,148.630
C07033=1170.785,335.653,-75.690,-176.461,8.413,148.629
C07034=1170.790,335.406,-75.657,-176.463,8.409,148.629
C07035=1170.794,335.158,-75.625,-176.466,8.406,148.629
C07036=1170.798,334.910,-75.592,-176.468,8.403,148.629
C07037=1170.802,334.662,-75.559,-176.471,8.399,148.629
C07038=1170.806,334.414,-75.527,-176.473,8.396,148.629
C07039=1170.810,334.167,-75.494,-176.476,8.393,148.629
C07040=1170.814,333.918,-75.462,-176.478,8.389,148.628
C07041=1170.818,333.671,-75.429,-176.481,8.386,148.628
C07042=1170.822,333.422,-75.397,-176.483,8.383,148.628
C07043=1170.827,333.175,-75.364,-176.486,8.380,148.628
C07044=1170.831,332.927,-75.332,-176.489,8.376,148.628
C07045=1170.835,332.680,-75.299,-176.491,8.372,148.628
C07046=1170.839,332.431,-75.266,-176.493,8.369,148.627
C07047=1170.843,332.184,-75.234,-176.496,8.366,148.627
C07048=1170.847,331.935,-75.201,-176.498,8.363,148.627
C07049=1170.851,331.688,-75.169,-176.500,8.360,148.627
C07050=1170.856,331.440,-75.137,-176.503,8.356,148.627
C07051=1170.860,331.192,-75.104,-176.505,8.353,148.627
C07052=1170.863,330.945,-75.072,-176.508,8.349,148.626
C07053=1170.868,330.696,-75.039,-176.511,8.346,148.626
C07054=1170.872,330.448,-75.008,-176.513,8.343,148.626
C07055=1170.876,330.201,-74.975,-176.516,8.340,148.626
C07056=1170.880,329.953,-74.943,-176.518,8.336,148.626
C07057=1170.885,329.705,-74.910,-176.520,8.333,148.626
C07058=1170.888,329.457,-74.878,-176.523,8.330,148.626
C07059=1170.892,329.209,-74.845,-176.525,8.327,148.625
C07060=1170.897,328.961,-74.813,-176.527,8.323,148.625
C07061=1170.901,328.713,-74.782,-176.531,8.320,148.625
C07062=1170.905,328.466,-74.749,-176.533,8.316,148.625
C07063=1170.909,328.218,-74.717,-176.535,8.313,148.625
C07064=1170.913,327.970,-74.685,-176.538,8.310,148.625
C07065=1170.918,327.722,-74.653,-176.540,8.307,148.625
C07066=1170.921,327.474,-74.621,-176.543,8.303,148.624
C07067=1170.926,327.226,-74.588,-176.545,8.300,148.624
C07068=1170.930,326.979,-74.556,-176.548,8.297,148.624
C07069=1170.934,326.730,-74.524,-176.550,8.294,148.624
C07070=1170.938,326.482,-74.492,-176.553,8.290,148.624
C07071=1170.942,326.234,-74.460,-176.555,8.287,148.624
C07072=1170.947,325.987,-74.428,-176.558,8.283,148.624
C07073=1170.950,325.739,-74.396,-176.560,8.280,148.624
C07074=1170.955,325.490,-74.364,-176.563,8.277,148.623
C07075=1170.959,325.243,-74.332,-176.565,8.274,148.623
C07076=1170.963,324.996,-74.300,-176.568,8.271,148.623
C07077=1170.967,324.747,-74.267,-176.570,8.268,148.623
C07078=1170.971,324.499,-74.235,-176.573,8.265,148.623
C07079=1170.975,324.252,-74.204,-176.575,8.261,148.623
C07080=1170.980,324.004,-74.171,-176.577,8.258,148.623
C07081=1170.983,323.756,-74.140,-176.581,8.254,148.623
C07082=1170.988,323.508,-74.108,-176.583,8.251,148.622
C07083=1170.992,323.259,-74.076,-176.586,8.248,148.622
C07084=1170.996,323.011,-74.045,-176.588,8.245,148.622
C07085=1171.000,322.764,-74.013,-176.590,8.241,148.622
C07086=1171.004,322.516,-73.981,-176.593,8.238,148.622
C07087=1171.008,322.267,-73.949,-176.595,8.235,148.622
C07088=1171.013,322.020,-73.917,-176.598,8.232,148.622
C07089=1171.016,321.772,-73.885,-176.600,8.229,148.622
C07090=1171.021,321.525,-73.854,-176.603,8.226,148.622
C07091=1171.025,321.276,-73.821,-176.605,8.222,148.621
C07092=1171.029,321.028,-73.790,-176.608,8.219,148.621
C07093=1171.034,320.780,-73.759,-176.610,8.216,148.621
C07094=1171.037,320.532,-73.727,-176.613,8.212,148.621
C07095=1171.042,320.284,-73.695,-176.616,8.209,148.621
C07096=1171.046,320.037,-73.663,-176.618,8.206,148.621
C07097=1171.050,319.788,-73.632,-176.621,8.203,148.621
C07098=1171.054,319.541,-73.601,-176.623,8.199,148.621
C07099=1171.058,319.293,-73.569,-176.626,8.196,148.621
C07100=1171.062,319.045,-73.537,-176.628,8.193,148.620
C07101=1171.067,318.796,-73.505,-176.631,8.190,148.620
C07102=1171.071,318.548,-73.474,-176.633,8.187,148.620
C07103=1171.075,318.301,-73.442,-176.635,8.184,148.620
C07104=1171.079,318.052,-73.411,-176.638,8.181,148.620
C07105=1171.083,317.805,-73.380,-176.640,8.177,148.620
C07106=1171.087,317.557,-73.348,-176.643,8.174,148.620
C07107=1171.092,317.309,-73.317,-176.645,8.171,148.620
C07108=1171.095,317.061,-73.285,-176.648,8.168,148.620
C07109=1171.100,316.813,-73.254,-176.651,8.165,148.620
C07110=1171.104,316.565,-73.222,-176.653,8.162,148.620
C07111=1171.109,316.317,-73.190,-176.656,8.158,148.619
C07112=1171.113,316.069,-73.159,-176.659,8.155,148.619
C07113=1171.117,315.821,-73.128,-176.661,8.151,148.619
C07114=1171.121,315.573,-73.097,-176.664,8.148,148.619
C07115=1171.125,315.325,-73.065,-176.666,8.145,148.619
C07116=1171.129,315.077,-73.034,-176.669,8.142,148.619
C07117=1171.134,314.829,-73.003,-176.671,8.139,148.619
C07118=1171.138,314.581,-72.971,-176.674,8.136,148.619
C07119=1171.142,314.304,-72.937,-176.677,8.133,148.619
C07120=1171.147,314.027,-72.902,-176.679,8.129,148.619
C07121=1171.152,313.750,-72.867,-176.682,8.126,148.619
C07122=1171.156,313.473,-72.832,-176.685,8.122,148.618
C07123=1171.160,313.225,-72.801,-176.688,8.119,148.618
C07124=1171.165,312.977,-72.770,-176.690,8.115,148.618
C07125=1171.169,312.729,-72.739,-176.693,8.112,148.618
C07126=1171.173,312.481,-72.707,-176.695,8.109,148.618
C07127=1171.177,312.233,-72.676,-176.698,8.106,148.618
C07128=1171.182,311.985,-72.645,-176.701,8.103,148.618
C07129=1171.186,311.737,-72.614,-176.703,8.100,148.618
C07130=1171.190,311.489,-72.583,-176.706,8.097,148.618
C07131=1171.194,311.241,-72.552,-176.708,8.093,148.618
C07132=1171.198,310.993,-72.520,-176.711,8.091,148.618
C07133=1171.202,310.745,-72.490,-176.713,8.087,148.617
C07134=1171.207,310.497,-72.459,-176.716,8.084,148.617
C07135=1171.211,310.248,-72.428,-176.718,8.081,148.617
C07136=1171.215,310.001,-72.397,-176.721,8.078,148.617
C07137=1171.219,309.752,-72.365,-176.723,8.075,148.617
C07138=1171.224,309.505,-72.335,-176.726,8.072,148.617
C07139=1171.228,309.257,-72.304,-176.728,8.069,148.617
C07140=1171.232,309.008,-72.273,-176.731,8.065,148.617
C07141=1171.236,308.760,-72.243,-176.733,8.062,148.617
C07142=1171.240,308.513,-72.211,-176.736,8.059,148.617
C07143=1171.244,308.264,-72.180,-176.738,8.056,148.617
C07144=1171.249,308.016,-72.149,-176.741,8.053,148.617
C07145=1171.253,307.769,-72.119,-176.743,8.050,148.617
C07146=1171.257,307.520,-72.088,-176.746,8.047,148.617
C07147=1171.262,307.272,-72.057,-176.749,8.044,148.617
C07148=1171.266,307.024,-72.026,-176.751,8.041,148.616
C07149=1171.269,306.776,-71.996,-176.754,8.038,148.616
C07150=1171.274,306.528,-71.965,-176.756,8.034,148.616
C07151=1171.279,306.280,-71.934,-176.759,8.031,148.616
C07152=1171.283,306.031,-71.903,-176.762,8.028,148.616
C07153=1171.287,305.783,-71.873,-176.764,8.025,148.616
C07154=1171.291,305.536,-71.842,-176.767,8.022,148.616
C07155=1171.296,305.288,-71.811,-176.769,8.019,148.616
C07156=1171.299,305.039,-71.781,-176.772,8.016,148.616
C07157=1171.304,304.791,-71.750,-176.774,8.013,148.616
C07158=1171.308,304.543,-71.719,-176.777,8.010,148.616
C07159=1171.312,304.296,-71.689,-176.779,8.007,148.616
C07160=1171.316,304.047,-71.658,-176.782,8.004,148.616
C07161=1171.321,303.799,-71.627,-176.784,8.000,148.616
C07162=1171.325,303.551,-71.597,-176.787,7.997,148.616
C07163=1171.329,303.303,-71.566,-176.790,7.994,148.616
C07164=1171.334,303.054,-71.536,-176.792,7.991,148.616
C07165=1171.337,302.807,-71.506,-176.795,7.988,148.616
C07166=1171.342,302.559,-71.475,-176.798,7.985,148.616
C07167=1171.346,302.311,-71.445,-176.800,7.982,148.615
C07168=1171.351,302.063,-71.414,-176.803,7.979,148.615
C07169=1171.355,301.814,-71.384,-176.805,7.976,148.615
C07170=1171.359,301.566,-71.354,-176.808,7.973,148.615
C07171=1171.363,301.318,-71.323,-176.810,7.970,148.615
C07172=1171.367,301.070,-71.293,-176.813,7.967,148.615
C07173=1171.372,300.822,-71.263,-176.815,7.963,148.615
C07174=1171.375,300.574,-71.232,-176.818,7.960,148.615
C07175=1171.380,300.326,-71.201,-176.821,7.957,148.615
C07176=1171.384,300.078,-71.171,-176.823,7.954,148.615
C07177=1171.389,299.829,-71.141,-176.826,7.951,148.615
C07178=1171.393,299.582,-71.111,-176.829,7.948,148.615
C07179=1171.397,299.333,-71.080,-176.831,7.945,148.615
C07180=1171.401,299.085,-71.050,-176.834,7.942,148.615
C07181=1171.406,298.837,-71.020,-176.836,7.939,148.615
C07182=1171.410,298.589,-70.990,-176.838,7.936,148.615
C07183=1171.414,298.341,-70.959,-176.841,7.933,148.615
C07184=1171.418,298.093,-70.929,-176.844,7.930,148.615
C07185=1171.423,297.844,-70.899,-176.846,7.927,148.615
C07186=1171.426,297.596,-70.869,-176.849,7.924,148.615
C07187=1171.431,297.348,-70.839,-176.851,7.921,148.615
C07188=1171.435,297.100,-70.808,-176.854,7.918,148.615
C07189=1171.439,296.851,-70.779,-176.856,7.915,148.615
C07190=1171.444,296.604,-70.748,-176.859,7.912,148.615
C07191=1171.448,296.355,-70.719,-176.862,7.909,148.615
C07192=1171.452,296.108,-70.688,-176.865,7.906,148.615
C07193=1171.457,295.859,-70.658,-176.867,7.903,148.614
C07194=1171.461,295.611,-70.628,-176.870,7.900,148.615
C07195=1171.465,295.363,-70.599,-176.872,7.897,148.615
C07196=1171.469,295.114,-70.568,-176.875,7.894,148.615
C07197=1171.473,294.866,-70.538,-176.877,7.890,148.614
C07198=1171.477,294.618,-70.509,-176.880,7.887,148.614
C07199=1171.482,294.370,-70.478,-176.883,7.884,148.614
C07200=1171.486,294.122,-70.449,-176.885,7.882,148.615
C07201=1171.490,293.874,-70.418,-176.887,7.879,148.614
C07202=1171.495,293.625,-70.388,-176.890,7.876,148.614
C07203=1171.499,293.377,-70.359,-176.893,7.873,148.614
C07204=1171.503,293.130,-70.329,-176.896,7.870,148.614
C07205=1171.507,292.881,-70.299,-176.898,7.867,148.614
C07206=1171.512,292.633,-70.269,-176.901,7.864,148.614
C07207=1171.516,292.384,-70.240,-176.903,7.861,148.614
C07208=1171.520,292.137,-70.210,-176.906,7.858,148.614
C07209=1171.524,291.889,-70.180,-176.908,7.855,148.614
C07210=1171.529,291.640,-70.151,-176.911,7.852,148.614
C07211=1171.533,291.392,-70.121,-176.914,7.849,148.614
C07212=1171.537,291.144,-70.090,-176.917,7.846,148.614
C07213=1171.542,290.896,-70.061,-176.919,7.843,148.614
C07214=1171.546,290.648,-70.032,-176.921,7.840,148.614
C07215=1171.550,290.399,-70.002,-176.924,7.837,148.614
C07216=1171.555,290.151,-69.972,-176.927,7.834,148.614
C07217=1171.559,289.903,-69.942,-176.929,7.831,148.614
C07218=1171.563,289.655,-69.912,-176.932,7.828,148.614
C07219=1171.567,289.406,-69.883,-176.934,7.825,148.614
C07220=1171.571,289.158,-69.854,-176.937,7.822,148.614
C07221=1171.575,288.910,-69.824,-176.940,7.819,148.614
C07222=1171.580,288.662,-69.795,-176.942,7.816,148.614
C07223=1171.585,288.388,-69.762,-176.945,7.813,148.614
C07224=1171.590,288.112,-69.729,-176.948,7.810,148.614
C07225=1171.595,287.837,-69.696,-176.951,7.806,148.614
C07226=1171.599,287.562,-69.664,-176.954,7.803,148.614
C07227=1171.603,287.314,-69.634,-176.956,7.800,148.614
C07228=1171.607,287.066,-69.605,-176.959,7.797,148.614
C07229=1171.613,286.818,-69.575,-176.962,7.794,148.614
C07230=1171.617,286.570,-69.546,-176.965,7.791,148.614
C07231=1171.621,286.321,-69.516,-176.966,7.789,148.614
C07232=1171.625,286.073,-69.487,-176.969,7.786,148.614
C07233=1171.629,285.825,-69.457,-176.972,7.783,148.614
C07234=1171.633,285.577,-69.428,-176.974,7.780,148.614
C07235=1171.638,285.328,-69.398,-176.977,7.777,148.614
C07236=1171.642,285.080,-69.370,-176.980,7.774,148.614
C07237=1171.647,284.832,-69.341,-176.982,7.770,148.614
C07238=1171.651,284.584,-69.311,-176.985,7.767,148.614
C07239=1171.655,284.335,-69.282,-176.988,7.765,148.614
C07240=1171.659,284.087,-69.252,-176.990,7.762,148.614
C07241=1171.664,283.839,-69.223,-176.993,7.759,148.614
C07242=1171.668,283.590,-69.194,-176.995,7.756,148.614
C07243=1171.672,283.342,-69.165,-176.998,7.753,148.614
C07244=1171.676,283.094,-69.136,-177.000,7.750,148.614
C07245=1171.680,282.846,-69.107,-177.003,7.747,148.614
C07246=1171.685,282.598,-69.077,-177.006,7.744,148.614
C07247=1171.689,282.349,-69.048,-177.008,7.742,148.614
C07248=1171.693,282.101,-69.019,-177.011,7.739,148.614
C07249=1171.698,281.853,-68.990,-177.014,7.736,148.614
C07250=1171.702,281.605,-68.960,-177.016,7.733,148.614
C07251=1171.707,281.356,-68.932,-177.019,7.730,148.615
C07252=1171.711,281.108,-68.902,-177.021,7.727,148.614
C07253=1171.715,280.861,-68.874,-177.024,7.724,148.614
C07254=1171.720,280.612,-68.845,-177.027,7.721,148.614
C07255=1171.724,280.363,-68.816,-177.029,7.719,148.614
C07256=1171.728,280.114,-68.787,-177.032,7.716,148.615
C07257=1171.732,279.866,-68.757,-177.034,7.713,148.615
C07258=1171.737,279.619,-68.728,-177.037,7.710,148.615
C07259=1171.741,279.370,-68.700,-177.040,7.707,148.615
C07260=1171.745,279.122,-68.671,-177.043,7.704,148.615
C07261=1171.750,278.873,-68.642,-177.045,7.701,148.615
C07262=1171.754,278.625,-68.613,-177.047,7.698,148.615
C07263=1171.758,278.377,-68.584,-177.050,7.695,148.615
C07264=1171.762,278.129,-68.555,-177.053,7.693,148.615
C07265=1171.767,277.881,-68.526,-177.055,7.690,148.615
C07266=1171.772,277.632,-68.497,-177.058,7.687,148.615
C07267=1171.775,277.384,-68.469,-177.061,7.684,148.615
C07268=1171.779,277.135,-68.440,-177.063,7.681,148.615
C07269=1171.785,276.887,-68.412,-177.066,7.678,148.615
C07270=1171.789,276.639,-68.382,-177.068,7.676,148.615
C07271=1171.792,276.390,-68.354,-177.071,7.673,148.615
C07272=1171.797,276.143,-68.325,-177.074,7.670,148.615
C07273=1171.802,275.894,-68.296,-177.077,7.667,148.615
C07274=1171.805,275.646,-68.267,-177.078,7.664,148.615
C07275=1171.810,275.398,-68.239,-177.081,7.661,148.615
C07276=1171.815,275.149,-68.210,-177.084,7.658,148.615
C07277=1171.818,274.901,-68.181,-177.087,7.655,148.615
C07278=1171.823,274.653,-68.153,-177.089,7.652,148.615
C07279=1171.827,274.404,-68.125,-177.092,7.649,148.615
C07280=1171.831,274.156,-68.095,-177.094,7.647,148.615
C07281=1171.836,273.908,-68.067,-177.097,7.644,148.615
C07282=1171.840,273.659,-68.039,-177.100,7.641,148.615
C07283=1171.844,273.411,-68.009,-177.103,7.638,148.615
C07284=1171.849,273.163,-67.982,-177.105,7.635,148.615
C07285=1171.853,272.914,-67.953,-177.107,7.633,148.616
C07286=1171.858,272.666,-67.924,-177.110,7.630,148.616
C07287=1171.862,272.418,-67.896,-177.113,7.627,148.616
C07288=1171.866,272.169,-67.867,-177.116,7.624,148.616
C07289=1171.870,271.921,-67.839,-177.118,7.621,148.616
C07290=1171.875,271.672,-67.810,-177.121,7.619,148.616
C07291=1171.879,271.424,-67.783,-177.123,7.616,148.616
C07292=1171.884,271.175,-67.754,-177.126,7.613,148.616
C07293=1171.888,270.928,-67.725,-177.129,7.610,148.616
C07294=1171.892,270.679,-67.697,-177.132,7.607,148.616
C07295=1171.896,270.431,-67.668,-177.134,7.604,148.616
C07296=1171.901,270.182,-67.640,-177.137,7.602,148.616
C07297=1171.905,269.934,-67.612,-177.139,7.599,148.616
C07298=1171.910,269.686,-67.584,-177.142,7.596,148.616
C07299=1171.914,269.437,-67.555,-177.145,7.593,148.616
C07300=1171.919,269.189,-67.527,-177.147,7.591,148.616
C07301=1171.923,268.940,-67.499,-177.150,7.588,148.616
C07302=1171.928,268.692,-67.471,-177.152,7.585,148.616
C07303=1171.931,268.444,-67.442,-177.155,7.582,148.617
C07304=1171.937,268.195,-67.414,-177.158,7.579,148.617
C07305=1171.940,267.947,-67.386,-177.160,7.577,148.617
C07306=1171.945,267.699,-67.358,-177.163,7.574,148.617
C07307=1171.949,267.450,-67.329,-177.166,7.571,148.617
C07308=1171.953,267.202,-67.302,-177.168,7.568,148.617
C07309=1171.958,266.953,-67.273,-177.171,7.565,148.617
C07310=1171.962,266.705,-67.245,-177.173,7.563,148.617
C07311=1171.966,266.457,-67.217,-177.176,7.560,148.617
